// TIA Portal V20 export
DATA_BLOCK "HmiInterface"   // DB90
{ DB_Accessible_From_OPC_UA := 'FALSE' }
AUTHOR : ERsystem_FA2_DH. Kim
// stored: Access Published, DBAccessibleFromOPCUA false, DBAccessibleFromWebserver false, MemoryReserve 100, Namespace Unit1.Em4
   VAR
      em : "LAF_typeEmInterface";
      cm : Struct
         softCam : "Unit1.type_emRelations_em4_SoftCam";
         brakeTest : Struct
            anodeMainPnP1AxisZ : "LER_typeBrakeTestEmInterface";
            anodeMainPnP2AxisZ : "LER_typeBrakeTestEmInterface";
         END_STRUCT;
      END_STRUCT;
      mainPnP : Struct
         jobs { S7_SetPoint := 'True'} : "LAF_typeJobsInterface";
         sequence { S7_SetPoint := 'True'} : "LAF_typeSequenceInterface";
      END_STRUCT;
      alignTable : Struct
         jobs { S7_SetPoint := 'True'} : "LAF_typeJobsInterface";
         sequence { S7_SetPoint := 'True'} : "LAF_typeSequenceInterface";
      END_STRUCT;
      ngPnP : Struct
         jobs { S7_SetPoint := 'True'} : "LAF_typeJobsInterface";
         sequence { S7_SetPoint := 'True'} : "LAF_typeSequenceInterface";
      END_STRUCT;
      gaugeRnR : Struct
         jobs { S7_SetPoint := 'True'} : "LAF_typeJobsInterface";
         sequence { S7_SetPoint := 'True'} : "LAF_typeSequenceInterface";
      END_STRUCT;
      anodeNgCount : "LER_typeAlarmCounterInterface";
      cmPnp1stAnodeDetect { S7_SetPoint := 'True'} : "LBC_typeDigitalSignalInterface";
      cmPnp2ndAnodeDetect { S7_SetPoint := 'True'} : "LBC_typeDigitalSignalInterface";
      cmAnodeAlignTableElectrodeDetect { S7_SetPoint := 'True'} : "LBC_typeDigitalSignalInterface";
      cmAnodeNgPnpElectrodeDetect { S7_SetPoint := 'True'} : "LBC_typeDigitalSignalInterface";
      cmAnodeNgBoxFullSensorDetect { S7_SetPoint := 'True'} : "LBC_typeDigitalSignalInterface";
      cmAnodeNgBoxDetect { S7_SetPoint := 'True'} : "LBC_typeDigitalSignalInterface";
   END_VAR
   VAR RETAIN
      cmAnodeMainPnP1AxisX : "LBC_typeAxis64PosInterface";
      cmAnodeMainPnP2AxisX : "LBC_typeAxis64PosInterface";
      cmAnodeMainPnP1AxisY : "LBC_typeAxis64PosInterface";
      cmAnodeMainPnP1AxisZ : "LBC_typeAxis64PosInterface";
      cmAnodeMainPnP2AxisZ : "LBC_typeAxis64PosInterface";
      cmAnodeAlignTableAxisX : "LBC_typeAxis64PosInterface";
      cmAnodeAlignTableAxisY1 : "LBC_typeAxis64PosInterface";
      cmAnodeAlignTableAxisY2 : "LBC_typeAxis64PosInterface";
   END_VAR
   VAR
      cmAnodeMainPnP1RotaryCwCcw : "LBC_typeTwoWayActuatorInterface";
      cmAnodeMainPnP1SuctionPlateVacuum : "LBC_typeTwoWayActuatorInterface";
      cmAnodeMainPnP2SuctionPlateVacuum : "LBC_typeTwoWayActuatorInterface";
      cmAnodeAlignTableSuctionPlateVacuum : "LBC_typeTwoWayActuatorInterface";
      cmAnodeGlassCleaning : "LBC_typeTwoWayActuatorInterface";
      cmAnodeNgPnpUpDown : "LBC_typeTwoWayActuatorInterface";
      cmAnodeNgPnp1stFwdBwd : "LBC_typeTwoWayActuatorInterface";
      cmAnodeNgPnp2ndFwdBwd { S7_SetPoint := 'True'} : "LBC_typeTwoWayActuatorInterface";
      cmAnodeMaintenanceMovingFixFrontRearFwdBwd : "LBC_typeTwoWayActuatorInterface";
      cmAnodeNgBoxLiftUpDown { S7_SetPoint := 'True'} : "LBC_typeTwoWayActuatorInterface";
      cmAnodeNgBoxLockUpDown { S7_SetPoint := 'True'} : "LBC_typeTwoWayActuatorInterface";
      cmAnodeNgPnpVaccum : "LBC_typeTwoWayActuatorInterface";
      cmAnodeConveyorCoverFwdBwd { S7_SetPoint := 'True'} : "LBC_typeTwoWayActuatorInterface";
      cmAnodeConveyorPickUpBlower { S7_SetPoint := 'True'} : "LBC_typeTwoWayActuatorInterface";
      cmAlignVisionControllerInterface : "LER_typeVisionInterface";
      AlignVisionConversion : "LER_typeVisionAlignResultData";
      AlignMoveCalibration : "LER_typeAlignMoveCalibrationInterface";
      AlignThetaCalibration { S7_SetPoint := 'True'} : "LER_typeAlignThetaCalibrationInterface";
      AlignVisionHistory : "LER_typeVisionHistory";
      AlignSyncMove : "LER_typeAlignSyncMoveInterface";
      AlignCalibration : "LER_typeAlignCalibrationInterface";
   END_VAR
   VAR RETAIN
      GaugeRnR1Align : "LER_typeCount";
   END_VAR
   VAR
      GaugeRnR1Stack : "LER_typeCount";
      GaugeRnR3Align : "LER_typeCount";
      intCondition : Struct
         Axis_05 { S7_SetPoint := 'True'} : "LER.typeAxisIntlockAll";   // AnodeMainPnP1AxisX
         Axis_06 { S7_SetPoint := 'True'} : "LER.typeAxisIntlockAll";   // AnodeMainPnP2AxisX
         Axis_11 { S7_SetPoint := 'True'} : "LER.typeAxisIntlockAll";   // AnodeMainPnP1AxisY
         Axis_12 { S7_SetPoint := 'True'} : "LER.typeAxisIntlockAll";   // AnodeMainPnP1AxisZ
         Axis_14 { S7_SetPoint := 'True'} : "LER.typeAxisIntlockAll";   // AnodeMainPnP2AxisZ
         Axis_15 { S7_SetPoint := 'True'} : "LER.typeAxisIntlockAll";   // AnodeAlignTableAxisX
         Axis_16 { S7_SetPoint := 'True'} : "LER.typeAxisIntlockAll";   // AnodeAlignTableAxisY1
         Axis_17 { S7_SetPoint := 'True'} : "LER.typeAxisIntlockAll";   // AnodeAlignTableAxisY2
         Actuator_13 { S7_SetPoint := 'True'} : "LER.typeAxisActuatorCondition";   // AnodeNgBoxLiftUpDown
         Actuator_14 { S7_SetPoint := 'True'} : "LER.typeAxisActuatorCondition";   // SP
         Actuator_15 { S7_SetPoint := 'True'} : "LER.typeAxisActuatorCondition";   // AnodeNgBoxLockUpDown
         Actuator_16 { S7_SetPoint := 'True'} : "LER.typeAxisActuatorCondition";   // AnodeMaintenanceMovingFixFrontFwdBwd
         Actuator_17 { S7_SetPoint := 'True'} : "LER.typeAxisActuatorCondition";   // AnodeGlassCleaning
         Actuator_18 { S7_SetPoint := 'True'} : "LER.typeAxisActuatorCondition";   // AnodeNgPnp1stFwdBwd
         Actuator_19 { S7_SetPoint := 'True'} : "LER.typeAxisActuatorCondition";   // AnodeNgPnpUpDown
         Actuator_20 { S7_SetPoint := 'True'} : "LER.typeAxisActuatorCondition";   // SP
         Actuator_21 { S7_SetPoint := 'True'} : "LER.typeAxisActuatorCondition";   // AnodeMainPnP1RotaryCwCcw
         Actuator_22 { S7_SetPoint := 'True'} : "LER.typeAxisActuatorCondition";   // AnodeNgPnp2ndFwdBwd
      END_STRUCT;
   END_VAR
BEGIN
   em.interlinkMode.link := FALSE;
   em.interlinkMode.unlink := FALSE;
   em.interlinkMode.isLinked := TRUE;
   em.commands.enable := FALSE;
   em.commands.acknowledge := FALSE;
   em.commands.disableAlarms := FALSE;
   em.commands.activateSimulation := FALSE;
   em.commands.home := FALSE;
   em.commands.moveToInitialPosition := FALSE;
   em.commands.directModeControl := 16#0000_0001;
   em.commands.directStateControl := 16#0000_0004;
   em.status.enabled := TRUE;
   em.status.acknowledgeActive := FALSE;
   em.status.alarmsDisabled := FALSE;
   em.status.simulationActive := TRUE;
   em.status.safetyReleased := TRUE;
   em.status.initialized := FALSE;
   em.status.homed := FALSE;
   em.status.safeState := FALSE;
   em.status.stateComplete := FALSE;
   em.alarms.error := FALSE;
   em.alarms.warning := FALSE;
   em.alarms.info := FALSE;
   em.alarms.home := FALSE;
   cm.softCam.anodeMainPnP1AxisX.reelCutConveyerPos.inPos := TRUE;
   cm.softCam.anodeMainPnP1AxisX.reelCutConveyerPos.isBefore := FALSE;
   cm.softCam.anodeMainPnP1AxisX.reelCutConveyerPos.isAfter := FALSE;
   cm.softCam.anodeMainPnP1AxisX.alignTablePos.inPos := FALSE;
   cm.softCam.anodeMainPnP1AxisX.alignTablePos.isBefore := FALSE;
   cm.softCam.anodeMainPnP1AxisX.alignTablePos.isAfter := TRUE;
   cm.softCam.anodeMainPnP1AxisX.Pos2.inPos := FALSE;
   cm.softCam.anodeMainPnP1AxisX.Pos2.isBefore := FALSE;
   cm.softCam.anodeMainPnP1AxisX.Pos2.isAfter := TRUE;
   cm.softCam.anodeMainPnP1AxisX.Pos3.inPos := FALSE;
   cm.softCam.anodeMainPnP1AxisX.Pos3.isBefore := FALSE;
   cm.softCam.anodeMainPnP1AxisX.Pos3.isAfter := TRUE;
   cm.softCam.anodeMainPnP1AxisX.Pos4.inPos := FALSE;
   cm.softCam.anodeMainPnP1AxisX.Pos4.isBefore := FALSE;
   cm.softCam.anodeMainPnP1AxisX.Pos4.isAfter := TRUE;
   cm.softCam.anodeMainPnP1AxisX.Pos5.inPos := FALSE;
   cm.softCam.anodeMainPnP1AxisX.Pos5.isBefore := FALSE;
   cm.softCam.anodeMainPnP1AxisX.Pos5.isAfter := TRUE;
   cm.softCam.anodeMainPnP1AxisX.Pos6.inPos := FALSE;
   cm.softCam.anodeMainPnP1AxisX.Pos6.isBefore := FALSE;
   cm.softCam.anodeMainPnP1AxisX.Pos6.isAfter := TRUE;
   cm.softCam.anodeMainPnP1AxisX.Pos7.inPos := FALSE;
   cm.softCam.anodeMainPnP1AxisX.Pos7.isBefore := FALSE;
   cm.softCam.anodeMainPnP1AxisX.Pos7.isAfter := TRUE;
   cm.softCam.anodeMainPnP1AxisX.Pos8.inPos := FALSE;
   cm.softCam.anodeMainPnP1AxisX.Pos8.isBefore := FALSE;
   cm.softCam.anodeMainPnP1AxisX.Pos8.isAfter := TRUE;
   cm.softCam.anodeMainPnP1AxisX.Pos9.inPos := FALSE;
   cm.softCam.anodeMainPnP1AxisX.Pos9.isBefore := FALSE;
   cm.softCam.anodeMainPnP1AxisX.Pos9.isAfter := TRUE;
   cm.softCam.anodeMainPnP1AxisX.Pos10.inPos := FALSE;
   cm.softCam.anodeMainPnP1AxisX.Pos10.isBefore := FALSE;
   cm.softCam.anodeMainPnP1AxisX.Pos10.isAfter := TRUE;
   cm.softCam.anodeMainPnP1AxisX.Pos11.inPos := FALSE;
   cm.softCam.anodeMainPnP1AxisX.Pos11.isBefore := FALSE;
   cm.softCam.anodeMainPnP1AxisX.Pos11.isAfter := TRUE;
   cm.softCam.anodeMainPnP1AxisX.Pos12.inPos := FALSE;
   cm.softCam.anodeMainPnP1AxisX.Pos12.isBefore := FALSE;
   cm.softCam.anodeMainPnP1AxisX.Pos12.isAfter := TRUE;
   cm.softCam.anodeMainPnP1AxisX.Pos13.inPos := FALSE;
   cm.softCam.anodeMainPnP1AxisX.Pos13.isBefore := FALSE;
   cm.softCam.anodeMainPnP1AxisX.Pos13.isAfter := TRUE;
   cm.softCam.anodeMainPnP1AxisX.Pos14.inPos := FALSE;
   cm.softCam.anodeMainPnP1AxisX.Pos14.isBefore := FALSE;
   cm.softCam.anodeMainPnP1AxisX.Pos14.isAfter := TRUE;
   cm.softCam.anodeMainPnP1AxisX.Pos15.inPos := FALSE;
   cm.softCam.anodeMainPnP1AxisX.Pos15.isBefore := FALSE;
   cm.softCam.anodeMainPnP1AxisX.Pos15.isAfter := TRUE;
   cm.softCam.anodeMainPnP2AxisX.alignTablePos.inPos := TRUE;
   cm.softCam.anodeMainPnP2AxisX.alignTablePos.isBefore := FALSE;
   cm.softCam.anodeMainPnP2AxisX.alignTablePos.isAfter := FALSE;
   cm.softCam.anodeMainPnP2AxisX.stackTablePos.inPos := FALSE;
   cm.softCam.anodeMainPnP2AxisX.stackTablePos.isBefore := FALSE;
   cm.softCam.anodeMainPnP2AxisX.stackTablePos.isAfter := TRUE;
   cm.softCam.anodeMainPnP2AxisX.Pos2.inPos := FALSE;
   cm.softCam.anodeMainPnP2AxisX.Pos2.isBefore := FALSE;
   cm.softCam.anodeMainPnP2AxisX.Pos2.isAfter := TRUE;
   cm.softCam.anodeMainPnP2AxisX.Pos3.inPos := FALSE;
   cm.softCam.anodeMainPnP2AxisX.Pos3.isBefore := FALSE;
   cm.softCam.anodeMainPnP2AxisX.Pos3.isAfter := TRUE;
   cm.softCam.anodeMainPnP2AxisX.Pos4.inPos := FALSE;
   cm.softCam.anodeMainPnP2AxisX.Pos4.isBefore := FALSE;
   cm.softCam.anodeMainPnP2AxisX.Pos4.isAfter := TRUE;
   cm.softCam.anodeMainPnP2AxisX.Pos5.inPos := FALSE;
   cm.softCam.anodeMainPnP2AxisX.Pos5.isBefore := FALSE;
   cm.softCam.anodeMainPnP2AxisX.Pos5.isAfter := TRUE;
   cm.softCam.anodeMainPnP2AxisX.Pos6.inPos := FALSE;
   cm.softCam.anodeMainPnP2AxisX.Pos6.isBefore := FALSE;
   cm.softCam.anodeMainPnP2AxisX.Pos6.isAfter := TRUE;
   cm.softCam.anodeMainPnP2AxisX.Pos7.inPos := FALSE;
   cm.softCam.anodeMainPnP2AxisX.Pos7.isBefore := FALSE;
   cm.softCam.anodeMainPnP2AxisX.Pos7.isAfter := TRUE;
   cm.softCam.anodeMainPnP2AxisX.Pos8.inPos := FALSE;
   cm.softCam.anodeMainPnP2AxisX.Pos8.isBefore := FALSE;
   cm.softCam.anodeMainPnP2AxisX.Pos8.isAfter := TRUE;
   cm.softCam.anodeMainPnP2AxisX.Pos9.inPos := FALSE;
   cm.softCam.anodeMainPnP2AxisX.Pos9.isBefore := FALSE;
   cm.softCam.anodeMainPnP2AxisX.Pos9.isAfter := TRUE;
   cm.softCam.anodeMainPnP2AxisX.Pos10.inPos := FALSE;
   cm.softCam.anodeMainPnP2AxisX.Pos10.isBefore := FALSE;
   cm.softCam.anodeMainPnP2AxisX.Pos10.isAfter := TRUE;
   cm.softCam.anodeMainPnP2AxisX.Pos11.inPos := FALSE;
   cm.softCam.anodeMainPnP2AxisX.Pos11.isBefore := FALSE;
   cm.softCam.anodeMainPnP2AxisX.Pos11.isAfter := TRUE;
   cm.softCam.anodeMainPnP2AxisX.Pos12.inPos := FALSE;
   cm.softCam.anodeMainPnP2AxisX.Pos12.isBefore := FALSE;
   cm.softCam.anodeMainPnP2AxisX.Pos12.isAfter := TRUE;
   cm.softCam.anodeMainPnP2AxisX.Pos13.inPos := FALSE;
   cm.softCam.anodeMainPnP2AxisX.Pos13.isBefore := FALSE;
   cm.softCam.anodeMainPnP2AxisX.Pos13.isAfter := TRUE;
   cm.softCam.anodeMainPnP2AxisX.Pos14.inPos := FALSE;
   cm.softCam.anodeMainPnP2AxisX.Pos14.isBefore := FALSE;
   cm.softCam.anodeMainPnP2AxisX.Pos14.isAfter := TRUE;
   cm.softCam.anodeMainPnP2AxisX.Pos15.inPos := FALSE;
   cm.softCam.anodeMainPnP2AxisX.Pos15.isBefore := FALSE;
   cm.softCam.anodeMainPnP2AxisX.Pos15.isAfter := TRUE;
   cm.softCam.anodeMainPnP1AxisY.waitPos.inPos := TRUE;
   cm.softCam.anodeMainPnP1AxisY.waitPos.isBefore := FALSE;
   cm.softCam.anodeMainPnP1AxisY.waitPos.isAfter := FALSE;
   cm.softCam.anodeMainPnP1AxisY.Pos1.inPos := TRUE;
   cm.softCam.anodeMainPnP1AxisY.Pos1.isBefore := FALSE;
   cm.softCam.anodeMainPnP1AxisY.Pos1.isAfter := FALSE;
   cm.softCam.anodeMainPnP1AxisY.Pos2.inPos := TRUE;
   cm.softCam.anodeMainPnP1AxisY.Pos2.isBefore := FALSE;
   cm.softCam.anodeMainPnP1AxisY.Pos2.isAfter := FALSE;
   cm.softCam.anodeMainPnP1AxisY.Pos3.inPos := TRUE;
   cm.softCam.anodeMainPnP1AxisY.Pos3.isBefore := FALSE;
   cm.softCam.anodeMainPnP1AxisY.Pos3.isAfter := FALSE;
   cm.softCam.anodeMainPnP1AxisY.Pos4.inPos := TRUE;
   cm.softCam.anodeMainPnP1AxisY.Pos4.isBefore := FALSE;
   cm.softCam.anodeMainPnP1AxisY.Pos4.isAfter := FALSE;
   cm.softCam.anodeMainPnP1AxisY.Pos5.inPos := TRUE;
   cm.softCam.anodeMainPnP1AxisY.Pos5.isBefore := FALSE;
   cm.softCam.anodeMainPnP1AxisY.Pos5.isAfter := FALSE;
   cm.softCam.anodeMainPnP1AxisY.Pos6.inPos := TRUE;
   cm.softCam.anodeMainPnP1AxisY.Pos6.isBefore := FALSE;
   cm.softCam.anodeMainPnP1AxisY.Pos6.isAfter := FALSE;
   cm.softCam.anodeMainPnP1AxisY.Pos7.inPos := TRUE;
   cm.softCam.anodeMainPnP1AxisY.Pos7.isBefore := FALSE;
   cm.softCam.anodeMainPnP1AxisY.Pos7.isAfter := FALSE;
   cm.softCam.anodeMainPnP1AxisY.Pos8.inPos := TRUE;
   cm.softCam.anodeMainPnP1AxisY.Pos8.isBefore := FALSE;
   cm.softCam.anodeMainPnP1AxisY.Pos8.isAfter := FALSE;
   cm.softCam.anodeMainPnP1AxisY.Pos9.inPos := TRUE;
   cm.softCam.anodeMainPnP1AxisY.Pos9.isBefore := FALSE;
   cm.softCam.anodeMainPnP1AxisY.Pos9.isAfter := FALSE;
   cm.softCam.anodeMainPnP1AxisY.Pos10.inPos := TRUE;
   cm.softCam.anodeMainPnP1AxisY.Pos10.isBefore := FALSE;
   cm.softCam.anodeMainPnP1AxisY.Pos10.isAfter := FALSE;
   cm.softCam.anodeMainPnP1AxisY.Pos11.inPos := TRUE;
   cm.softCam.anodeMainPnP1AxisY.Pos11.isBefore := FALSE;
   cm.softCam.anodeMainPnP1AxisY.Pos11.isAfter := FALSE;
   cm.softCam.anodeMainPnP1AxisY.Pos12.inPos := TRUE;
   cm.softCam.anodeMainPnP1AxisY.Pos12.isBefore := FALSE;
   cm.softCam.anodeMainPnP1AxisY.Pos12.isAfter := FALSE;
   cm.softCam.anodeMainPnP1AxisY.Pos13.inPos := TRUE;
   cm.softCam.anodeMainPnP1AxisY.Pos13.isBefore := FALSE;
   cm.softCam.anodeMainPnP1AxisY.Pos13.isAfter := FALSE;
   cm.softCam.anodeMainPnP1AxisY.Pos14.inPos := TRUE;
   cm.softCam.anodeMainPnP1AxisY.Pos14.isBefore := FALSE;
   cm.softCam.anodeMainPnP1AxisY.Pos14.isAfter := FALSE;
   cm.softCam.anodeMainPnP1AxisY.Pos15.inPos := TRUE;
   cm.softCam.anodeMainPnP1AxisY.Pos15.isBefore := FALSE;
   cm.softCam.anodeMainPnP1AxisY.Pos15.isAfter := FALSE;
   cm.softCam.anodeMainPnP1AxisZ.upPos.inPos := FALSE;
   cm.softCam.anodeMainPnP1AxisZ.upPos.isBefore := FALSE;
   cm.softCam.anodeMainPnP1AxisZ.upPos.isAfter := TRUE;
   cm.softCam.anodeMainPnP1AxisZ.reelCutConveyerDownPos.inPos := TRUE;
   cm.softCam.anodeMainPnP1AxisZ.reelCutConveyerDownPos.isBefore := FALSE;
   cm.softCam.anodeMainPnP1AxisZ.reelCutConveyerDownPos.isAfter := FALSE;
   cm.softCam.anodeMainPnP1AxisZ.ailgnTableDownPos.inPos := TRUE;
   cm.softCam.anodeMainPnP1AxisZ.ailgnTableDownPos.isBefore := FALSE;
   cm.softCam.anodeMainPnP1AxisZ.ailgnTableDownPos.isAfter := FALSE;
   cm.softCam.anodeMainPnP1AxisZ.avoidPos.inPos := FALSE;
   cm.softCam.anodeMainPnP1AxisZ.avoidPos.isBefore := FALSE;
   cm.softCam.anodeMainPnP1AxisZ.avoidPos.isAfter := TRUE;
   cm.softCam.anodeMainPnP1AxisZ.Pos4.inPos := FALSE;
   cm.softCam.anodeMainPnP1AxisZ.Pos4.isBefore := FALSE;
   cm.softCam.anodeMainPnP1AxisZ.Pos4.isAfter := TRUE;
   cm.softCam.anodeMainPnP1AxisZ.Pos5.inPos := FALSE;
   cm.softCam.anodeMainPnP1AxisZ.Pos5.isBefore := FALSE;
   cm.softCam.anodeMainPnP1AxisZ.Pos5.isAfter := TRUE;
   cm.softCam.anodeMainPnP1AxisZ.Pos6.inPos := FALSE;
   cm.softCam.anodeMainPnP1AxisZ.Pos6.isBefore := FALSE;
   cm.softCam.anodeMainPnP1AxisZ.Pos6.isAfter := TRUE;
   cm.softCam.anodeMainPnP1AxisZ.Pos7.inPos := FALSE;
   cm.softCam.anodeMainPnP1AxisZ.Pos7.isBefore := FALSE;
   cm.softCam.anodeMainPnP1AxisZ.Pos7.isAfter := TRUE;
   cm.softCam.anodeMainPnP1AxisZ.Pos8.inPos := FALSE;
   cm.softCam.anodeMainPnP1AxisZ.Pos8.isBefore := FALSE;
   cm.softCam.anodeMainPnP1AxisZ.Pos8.isAfter := TRUE;
   cm.softCam.anodeMainPnP1AxisZ.Pos9.inPos := FALSE;
   cm.softCam.anodeMainPnP1AxisZ.Pos9.isBefore := FALSE;
   cm.softCam.anodeMainPnP1AxisZ.Pos9.isAfter := TRUE;
   cm.softCam.anodeMainPnP1AxisZ.Pos10.inPos := FALSE;
   cm.softCam.anodeMainPnP1AxisZ.Pos10.isBefore := FALSE;
   cm.softCam.anodeMainPnP1AxisZ.Pos10.isAfter := TRUE;
   cm.softCam.anodeMainPnP1AxisZ.Pos11.inPos := FALSE;
   cm.softCam.anodeMainPnP1AxisZ.Pos11.isBefore := FALSE;
   cm.softCam.anodeMainPnP1AxisZ.Pos11.isAfter := TRUE;
   cm.softCam.anodeMainPnP1AxisZ.Pos12.inPos := FALSE;
   cm.softCam.anodeMainPnP1AxisZ.Pos12.isBefore := FALSE;
   cm.softCam.anodeMainPnP1AxisZ.Pos12.isAfter := TRUE;
   cm.softCam.anodeMainPnP1AxisZ.Pos13.inPos := FALSE;
   cm.softCam.anodeMainPnP1AxisZ.Pos13.isBefore := FALSE;
   cm.softCam.anodeMainPnP1AxisZ.Pos13.isAfter := TRUE;
   cm.softCam.anodeMainPnP1AxisZ.Pos14.inPos := FALSE;
   cm.softCam.anodeMainPnP1AxisZ.Pos14.isBefore := FALSE;
   cm.softCam.anodeMainPnP1AxisZ.Pos14.isAfter := TRUE;
   cm.softCam.anodeMainPnP1AxisZ.Pos15.inPos := FALSE;
   cm.softCam.anodeMainPnP1AxisZ.Pos15.isBefore := FALSE;
   cm.softCam.anodeMainPnP1AxisZ.Pos15.isAfter := TRUE;
   cm.softCam.anodeMainPnP2AxisZ.upPos.inPos := FALSE;
   cm.softCam.anodeMainPnP2AxisZ.upPos.isBefore := FALSE;
   cm.softCam.anodeMainPnP2AxisZ.upPos.isAfter := TRUE;
   cm.softCam.anodeMainPnP2AxisZ.ailgnTableDownPos.inPos := TRUE;
   cm.softCam.anodeMainPnP2AxisZ.ailgnTableDownPos.isBefore := FALSE;
   cm.softCam.anodeMainPnP2AxisZ.ailgnTableDownPos.isAfter := FALSE;
   cm.softCam.anodeMainPnP2AxisZ.stackTableDownPos.inPos := TRUE;
   cm.softCam.anodeMainPnP2AxisZ.stackTableDownPos.isBefore := FALSE;
   cm.softCam.anodeMainPnP2AxisZ.stackTableDownPos.isAfter := FALSE;
   cm.softCam.anodeMainPnP2AxisZ.avoidPos.inPos := FALSE;
   cm.softCam.anodeMainPnP2AxisZ.avoidPos.isBefore := FALSE;
   cm.softCam.anodeMainPnP2AxisZ.avoidPos.isAfter := TRUE;
   cm.softCam.anodeMainPnP2AxisZ.Pos4.inPos := FALSE;
   cm.softCam.anodeMainPnP2AxisZ.Pos4.isBefore := FALSE;
   cm.softCam.anodeMainPnP2AxisZ.Pos4.isAfter := TRUE;
   cm.softCam.anodeMainPnP2AxisZ.Pos5.inPos := FALSE;
   cm.softCam.anodeMainPnP2AxisZ.Pos5.isBefore := FALSE;
   cm.softCam.anodeMainPnP2AxisZ.Pos5.isAfter := TRUE;
   cm.softCam.anodeMainPnP2AxisZ.Pos6.inPos := FALSE;
   cm.softCam.anodeMainPnP2AxisZ.Pos6.isBefore := FALSE;
   cm.softCam.anodeMainPnP2AxisZ.Pos6.isAfter := TRUE;
   cm.softCam.anodeMainPnP2AxisZ.Pos7.inPos := FALSE;
   cm.softCam.anodeMainPnP2AxisZ.Pos7.isBefore := FALSE;
   cm.softCam.anodeMainPnP2AxisZ.Pos7.isAfter := TRUE;
   cm.softCam.anodeMainPnP2AxisZ.Pos8.inPos := FALSE;
   cm.softCam.anodeMainPnP2AxisZ.Pos8.isBefore := FALSE;
   cm.softCam.anodeMainPnP2AxisZ.Pos8.isAfter := TRUE;
   cm.softCam.anodeMainPnP2AxisZ.Pos9.inPos := FALSE;
   cm.softCam.anodeMainPnP2AxisZ.Pos9.isBefore := FALSE;
   cm.softCam.anodeMainPnP2AxisZ.Pos9.isAfter := TRUE;
   cm.softCam.anodeMainPnP2AxisZ.Pos10.inPos := FALSE;
   cm.softCam.anodeMainPnP2AxisZ.Pos10.isBefore := FALSE;
   cm.softCam.anodeMainPnP2AxisZ.Pos10.isAfter := TRUE;
   cm.softCam.anodeMainPnP2AxisZ.Pos11.inPos := FALSE;
   cm.softCam.anodeMainPnP2AxisZ.Pos11.isBefore := FALSE;
   cm.softCam.anodeMainPnP2AxisZ.Pos11.isAfter := TRUE;
   cm.softCam.anodeMainPnP2AxisZ.Pos12.inPos := FALSE;
   cm.softCam.anodeMainPnP2AxisZ.Pos12.isBefore := FALSE;
   cm.softCam.anodeMainPnP2AxisZ.Pos12.isAfter := TRUE;
   cm.softCam.anodeMainPnP2AxisZ.Pos13.inPos := FALSE;
   cm.softCam.anodeMainPnP2AxisZ.Pos13.isBefore := FALSE;
   cm.softCam.anodeMainPnP2AxisZ.Pos13.isAfter := TRUE;
   cm.softCam.anodeMainPnP2AxisZ.Pos14.inPos := FALSE;
   cm.softCam.anodeMainPnP2AxisZ.Pos14.isBefore := FALSE;
   cm.softCam.anodeMainPnP2AxisZ.Pos14.isAfter := TRUE;
   cm.softCam.anodeMainPnP2AxisZ.Pos15.inPos := FALSE;
   cm.softCam.anodeMainPnP2AxisZ.Pos15.isBefore := FALSE;
   cm.softCam.anodeMainPnP2AxisZ.Pos15.isAfter := TRUE;
   cm.softCam.anodeAlignTableAxisX.waitPos.inPos := TRUE;
   cm.softCam.anodeAlignTableAxisX.waitPos.isBefore := FALSE;
   cm.softCam.anodeAlignTableAxisX.waitPos.isAfter := FALSE;
   cm.softCam.anodeAlignTableAxisX.adjustPos.inPos := FALSE;
   cm.softCam.anodeAlignTableAxisX.adjustPos.isBefore := TRUE;
   cm.softCam.anodeAlignTableAxisX.adjustPos.isAfter := FALSE;
   cm.softCam.anodeAlignTableAxisX.Pos2.inPos := FALSE;
   cm.softCam.anodeAlignTableAxisX.Pos2.isBefore := FALSE;
   cm.softCam.anodeAlignTableAxisX.Pos2.isAfter := TRUE;
   cm.softCam.anodeAlignTableAxisX.Pos3.inPos := FALSE;
   cm.softCam.anodeAlignTableAxisX.Pos3.isBefore := FALSE;
   cm.softCam.anodeAlignTableAxisX.Pos3.isAfter := TRUE;
   cm.softCam.anodeAlignTableAxisX.Pos4.inPos := FALSE;
   cm.softCam.anodeAlignTableAxisX.Pos4.isBefore := FALSE;
   cm.softCam.anodeAlignTableAxisX.Pos4.isAfter := TRUE;
   cm.softCam.anodeAlignTableAxisX.Pos5.inPos := FALSE;
   cm.softCam.anodeAlignTableAxisX.Pos5.isBefore := FALSE;
   cm.softCam.anodeAlignTableAxisX.Pos5.isAfter := TRUE;
   cm.softCam.anodeAlignTableAxisX.Pos6.inPos := FALSE;
   cm.softCam.anodeAlignTableAxisX.Pos6.isBefore := FALSE;
   cm.softCam.anodeAlignTableAxisX.Pos6.isAfter := TRUE;
   cm.softCam.anodeAlignTableAxisX.Pos7.inPos := FALSE;
   cm.softCam.anodeAlignTableAxisX.Pos7.isBefore := FALSE;
   cm.softCam.anodeAlignTableAxisX.Pos7.isAfter := TRUE;
   cm.softCam.anodeAlignTableAxisX.Pos8.inPos := FALSE;
   cm.softCam.anodeAlignTableAxisX.Pos8.isBefore := FALSE;
   cm.softCam.anodeAlignTableAxisX.Pos8.isAfter := TRUE;
   cm.softCam.anodeAlignTableAxisX.Pos9.inPos := FALSE;
   cm.softCam.anodeAlignTableAxisX.Pos9.isBefore := FALSE;
   cm.softCam.anodeAlignTableAxisX.Pos9.isAfter := TRUE;
   cm.softCam.anodeAlignTableAxisX.Pos10.inPos := FALSE;
   cm.softCam.anodeAlignTableAxisX.Pos10.isBefore := TRUE;
   cm.softCam.anodeAlignTableAxisX.Pos10.isAfter := FALSE;
   cm.softCam.anodeAlignTableAxisX.Pos11.inPos := TRUE;
   cm.softCam.anodeAlignTableAxisX.Pos11.isBefore := FALSE;
   cm.softCam.anodeAlignTableAxisX.Pos11.isAfter := FALSE;
   cm.softCam.anodeAlignTableAxisX.Pos12.inPos := TRUE;
   cm.softCam.anodeAlignTableAxisX.Pos12.isBefore := FALSE;
   cm.softCam.anodeAlignTableAxisX.Pos12.isAfter := FALSE;
   cm.softCam.anodeAlignTableAxisX.Pos13.inPos := TRUE;
   cm.softCam.anodeAlignTableAxisX.Pos13.isBefore := FALSE;
   cm.softCam.anodeAlignTableAxisX.Pos13.isAfter := FALSE;
   cm.softCam.anodeAlignTableAxisX.Pos14.inPos := TRUE;
   cm.softCam.anodeAlignTableAxisX.Pos14.isBefore := FALSE;
   cm.softCam.anodeAlignTableAxisX.Pos14.isAfter := FALSE;
   cm.softCam.anodeAlignTableAxisX.Pos15.inPos := TRUE;
   cm.softCam.anodeAlignTableAxisX.Pos15.isBefore := FALSE;
   cm.softCam.anodeAlignTableAxisX.Pos15.isAfter := FALSE;
   cm.softCam.anodeAlignTableAxisY1.waitPos.inPos := TRUE;
   cm.softCam.anodeAlignTableAxisY1.waitPos.isBefore := FALSE;
   cm.softCam.anodeAlignTableAxisY1.waitPos.isAfter := FALSE;
   cm.softCam.anodeAlignTableAxisY1.adjustPos.inPos := FALSE;
   cm.softCam.anodeAlignTableAxisY1.adjustPos.isBefore := TRUE;
   cm.softCam.anodeAlignTableAxisY1.adjustPos.isAfter := FALSE;
   cm.softCam.anodeAlignTableAxisY1.Pos2.inPos := FALSE;
   cm.softCam.anodeAlignTableAxisY1.Pos2.isBefore := TRUE;
   cm.softCam.anodeAlignTableAxisY1.Pos2.isAfter := FALSE;
   cm.softCam.anodeAlignTableAxisY1.Pos3.inPos := FALSE;
   cm.softCam.anodeAlignTableAxisY1.Pos3.isBefore := TRUE;
   cm.softCam.anodeAlignTableAxisY1.Pos3.isAfter := FALSE;
   cm.softCam.anodeAlignTableAxisY1.Pos4.inPos := FALSE;
   cm.softCam.anodeAlignTableAxisY1.Pos4.isBefore := TRUE;
   cm.softCam.anodeAlignTableAxisY1.Pos4.isAfter := FALSE;
   cm.softCam.anodeAlignTableAxisY1.Pos5.inPos := FALSE;
   cm.softCam.anodeAlignTableAxisY1.Pos5.isBefore := TRUE;
   cm.softCam.anodeAlignTableAxisY1.Pos5.isAfter := FALSE;
   cm.softCam.anodeAlignTableAxisY1.Pos6.inPos := FALSE;
   cm.softCam.anodeAlignTableAxisY1.Pos6.isBefore := TRUE;
   cm.softCam.anodeAlignTableAxisY1.Pos6.isAfter := FALSE;
   cm.softCam.anodeAlignTableAxisY1.Pos7.inPos := FALSE;
   cm.softCam.anodeAlignTableAxisY1.Pos7.isBefore := FALSE;
   cm.softCam.anodeAlignTableAxisY1.Pos7.isAfter := TRUE;
   cm.softCam.anodeAlignTableAxisY1.Pos8.inPos := FALSE;
   cm.softCam.anodeAlignTableAxisY1.Pos8.isBefore := TRUE;
   cm.softCam.anodeAlignTableAxisY1.Pos8.isAfter := FALSE;
   cm.softCam.anodeAlignTableAxisY1.Pos9.inPos := FALSE;
   cm.softCam.anodeAlignTableAxisY1.Pos9.isBefore := FALSE;
   cm.softCam.anodeAlignTableAxisY1.Pos9.isAfter := TRUE;
   cm.softCam.anodeAlignTableAxisY1.Pos10.inPos := FALSE;
   cm.softCam.anodeAlignTableAxisY1.Pos10.isBefore := TRUE;
   cm.softCam.anodeAlignTableAxisY1.Pos10.isAfter := FALSE;
   cm.softCam.anodeAlignTableAxisY1.Pos11.inPos := TRUE;
   cm.softCam.anodeAlignTableAxisY1.Pos11.isBefore := FALSE;
   cm.softCam.anodeAlignTableAxisY1.Pos11.isAfter := FALSE;
   cm.softCam.anodeAlignTableAxisY1.Pos12.inPos := TRUE;
   cm.softCam.anodeAlignTableAxisY1.Pos12.isBefore := FALSE;
   cm.softCam.anodeAlignTableAxisY1.Pos12.isAfter := FALSE;
   cm.softCam.anodeAlignTableAxisY1.Pos13.inPos := TRUE;
   cm.softCam.anodeAlignTableAxisY1.Pos13.isBefore := FALSE;
   cm.softCam.anodeAlignTableAxisY1.Pos13.isAfter := FALSE;
   cm.softCam.anodeAlignTableAxisY1.Pos14.inPos := TRUE;
   cm.softCam.anodeAlignTableAxisY1.Pos14.isBefore := FALSE;
   cm.softCam.anodeAlignTableAxisY1.Pos14.isAfter := FALSE;
   cm.softCam.anodeAlignTableAxisY1.Pos15.inPos := TRUE;
   cm.softCam.anodeAlignTableAxisY1.Pos15.isBefore := FALSE;
   cm.softCam.anodeAlignTableAxisY1.Pos15.isAfter := FALSE;
   cm.softCam.anodeAlignTableAxisY2.waitPos.inPos := TRUE;
   cm.softCam.anodeAlignTableAxisY2.waitPos.isBefore := FALSE;
   cm.softCam.anodeAlignTableAxisY2.waitPos.isAfter := FALSE;
   cm.softCam.anodeAlignTableAxisY2.adjustPos.inPos := FALSE;
   cm.softCam.anodeAlignTableAxisY2.adjustPos.isBefore := TRUE;
   cm.softCam.anodeAlignTableAxisY2.adjustPos.isAfter := FALSE;
   cm.softCam.anodeAlignTableAxisY2.Pos2.inPos := TRUE;
   cm.softCam.anodeAlignTableAxisY2.Pos2.isBefore := FALSE;
   cm.softCam.anodeAlignTableAxisY2.Pos2.isAfter := FALSE;
   cm.softCam.anodeAlignTableAxisY2.Pos3.inPos := TRUE;
   cm.softCam.anodeAlignTableAxisY2.Pos3.isBefore := FALSE;
   cm.softCam.anodeAlignTableAxisY2.Pos3.isAfter := FALSE;
   cm.softCam.anodeAlignTableAxisY2.Pos4.inPos := TRUE;
   cm.softCam.anodeAlignTableAxisY2.Pos4.isBefore := FALSE;
   cm.softCam.anodeAlignTableAxisY2.Pos4.isAfter := FALSE;
   cm.softCam.anodeAlignTableAxisY2.Pos5.inPos := TRUE;
   cm.softCam.anodeAlignTableAxisY2.Pos5.isBefore := FALSE;
   cm.softCam.anodeAlignTableAxisY2.Pos5.isAfter := FALSE;
   cm.softCam.anodeAlignTableAxisY2.Pos6.inPos := TRUE;
   cm.softCam.anodeAlignTableAxisY2.Pos6.isBefore := FALSE;
   cm.softCam.anodeAlignTableAxisY2.Pos6.isAfter := FALSE;
   cm.softCam.anodeAlignTableAxisY2.Pos7.inPos := TRUE;
   cm.softCam.anodeAlignTableAxisY2.Pos7.isBefore := FALSE;
   cm.softCam.anodeAlignTableAxisY2.Pos7.isAfter := FALSE;
   cm.softCam.anodeAlignTableAxisY2.Pos8.inPos := TRUE;
   cm.softCam.anodeAlignTableAxisY2.Pos8.isBefore := FALSE;
   cm.softCam.anodeAlignTableAxisY2.Pos8.isAfter := FALSE;
   cm.softCam.anodeAlignTableAxisY2.Pos9.inPos := TRUE;
   cm.softCam.anodeAlignTableAxisY2.Pos9.isBefore := FALSE;
   cm.softCam.anodeAlignTableAxisY2.Pos9.isAfter := FALSE;
   cm.softCam.anodeAlignTableAxisY2.Pos10.inPos := FALSE;
   cm.softCam.anodeAlignTableAxisY2.Pos10.isBefore := TRUE;
   cm.softCam.anodeAlignTableAxisY2.Pos10.isAfter := FALSE;
   cm.softCam.anodeAlignTableAxisY2.Pos11.inPos := TRUE;
   cm.softCam.anodeAlignTableAxisY2.Pos11.isBefore := FALSE;
   cm.softCam.anodeAlignTableAxisY2.Pos11.isAfter := FALSE;
   cm.softCam.anodeAlignTableAxisY2.Pos12.inPos := TRUE;
   cm.softCam.anodeAlignTableAxisY2.Pos12.isBefore := FALSE;
   cm.softCam.anodeAlignTableAxisY2.Pos12.isAfter := FALSE;
   cm.softCam.anodeAlignTableAxisY2.Pos13.inPos := TRUE;
   cm.softCam.anodeAlignTableAxisY2.Pos13.isBefore := FALSE;
   cm.softCam.anodeAlignTableAxisY2.Pos13.isAfter := FALSE;
   cm.softCam.anodeAlignTableAxisY2.Pos14.inPos := TRUE;
   cm.softCam.anodeAlignTableAxisY2.Pos14.isBefore := FALSE;
   cm.softCam.anodeAlignTableAxisY2.Pos14.isAfter := FALSE;
   cm.softCam.anodeAlignTableAxisY2.Pos15.inPos := TRUE;
   cm.softCam.anodeAlignTableAxisY2.Pos15.isBefore := FALSE;
   cm.softCam.anodeAlignTableAxisY2.Pos15.isAfter := FALSE;
   cm.brakeTest.anodeMainPnP1AxisZ.commands.start := FALSE;
   cm.brakeTest.anodeMainPnP1AxisZ.commands.stop := FALSE;
   cm.brakeTest.anodeMainPnP1AxisZ.monitoring.error := FALSE;
   cm.brakeTest.anodeMainPnP1AxisZ.monitoring.ready := FALSE;
   cm.brakeTest.anodeMainPnP1AxisZ.monitoring.busy := FALSE;
   cm.brakeTest.anodeMainPnP1AxisZ.monitoring.complete := FALSE;
   cm.brakeTest.anodeMainPnP1AxisZ.monitoring.brakeSelected := FALSE;
   cm.brakeTest.anodeMainPnP1AxisZ.monitoring.brakeActive := FALSE;
   cm.brakeTest.anodeMainPnP1AxisZ.monitoring.brakeResult := FALSE;
   cm.brakeTest.anodeMainPnP1AxisZ.monitoring.brakeCompleted := FALSE;
   cm.brakeTest.anodeMainPnP1AxisZ.monitoring."step" := 0;
   cm.brakeTest.anodeMainPnP2AxisZ.commands.start := FALSE;
   cm.brakeTest.anodeMainPnP2AxisZ.commands.stop := FALSE;
   cm.brakeTest.anodeMainPnP2AxisZ.monitoring.error := FALSE;
   cm.brakeTest.anodeMainPnP2AxisZ.monitoring.ready := FALSE;
   cm.brakeTest.anodeMainPnP2AxisZ.monitoring.busy := FALSE;
   cm.brakeTest.anodeMainPnP2AxisZ.monitoring.complete := FALSE;
   cm.brakeTest.anodeMainPnP2AxisZ.monitoring.brakeSelected := FALSE;
   cm.brakeTest.anodeMainPnP2AxisZ.monitoring.brakeActive := FALSE;
   cm.brakeTest.anodeMainPnP2AxisZ.monitoring.brakeResult := FALSE;
   cm.brakeTest.anodeMainPnP2AxisZ.monitoring.brakeCompleted := FALSE;
   cm.brakeTest.anodeMainPnP2AxisZ.monitoring."step" := 0;
   mainPnP.jobs.commands.setJobNumber := 0;
   mainPnP.jobs.commands.reset := FALSE;
   mainPnP.jobs.status.activeJobNumber := 0;
   mainPnP.jobs.status.previousCycleJobNumber := 0;
   mainPnP.jobs.status.manualControlEnabled := FALSE;
   mainPnP.jobs.status.memoryJobTime := 16#0000_4EB7_0DCE_2E62;
   mainPnP.sequence.commands.setAutomaticMode := FALSE;
   mainPnP.sequence.commands.setSingleStepMode := FALSE;
   mainPnP.sequence.commands.off := FALSE;
   mainPnP.sequence.commands.initialize := FALSE;
   mainPnP.sequence.commands.start := FALSE;
   mainPnP.sequence.commands.immediateStop := FALSE;
   mainPnP.sequence.commands.hold := FALSE;
   mainPnP.sequence.commands.nextStep := FALSE;
   mainPnP.sequence.commands.interlockStepChange := FALSE;
   mainPnP.sequence.monitoring.automaticMode := TRUE;
   mainPnP.sequence.monitoring.singleStepMode := FALSE;
   mainPnP.sequence.monitoring.currentStep := 1;
   mainPnP.sequence.monitoring.nextStep := 1;
   mainPnP.sequence.monitoring.previousStep := 190;
   mainPnP.sequence.monitoring.currentStepSTRING := 'N/A';
   mainPnP.sequence.monitoring.nextStepSTRING := 'N/A';
   mainPnP.sequence.monitoring.previousStepSTRING := 'N/A';
   mainPnP.sequence.monitoring.inStepIdle := TRUE;
   mainPnP.sequence.monitoring.inStepStopped := FALSE;
   mainPnP.sequence.monitoring.seqActive := TRUE;
   mainPnP.sequence.monitoring.stepActive := TRUE;
   mainPnP.sequence.monitoring.stepComplete := FALSE;
   mainPnP.sequence.monitoring.executionEnabled := TRUE;
   mainPnP.sequence.monitoring.initRequired := FALSE;
   mainPnP.sequence.monitoring.stepChangeReleased := TRUE;
   mainPnP.sequence.monitoring.justSteppedPulse := FALSE;
   mainPnP.sequence.monitoring.manualControlEnabled := FALSE;
   mainPnP.sequence.monitoring.manualModeChangeEnabled := FALSE;
   mainPnP.sequence.monitoring.memoryStepTimer := 16#0000_4EB7_0DCD_6EA2;
   alignTable.jobs.commands.setJobNumber := 0;
   alignTable.jobs.commands.reset := FALSE;
   alignTable.jobs.status.activeJobNumber := 1;
   alignTable.jobs.status.previousCycleJobNumber := 1;
   alignTable.jobs.status.manualControlEnabled := FALSE;
   alignTable.jobs.status.memoryJobTime := 16#0000_4E8D_4592_AC24;
   alignTable.sequence.commands.setAutomaticMode := FALSE;
   alignTable.sequence.commands.setSingleStepMode := FALSE;
   alignTable.sequence.commands.off := FALSE;
   alignTable.sequence.commands.initialize := FALSE;
   alignTable.sequence.commands.start := FALSE;
   alignTable.sequence.commands.immediateStop := FALSE;
   alignTable.sequence.commands.hold := FALSE;
   alignTable.sequence.commands.nextStep := FALSE;
   alignTable.sequence.commands.interlockStepChange := FALSE;
   alignTable.sequence.monitoring.automaticMode := TRUE;
   alignTable.sequence.monitoring.singleStepMode := FALSE;
   alignTable.sequence.monitoring.currentStep := 160;
   alignTable.sequence.monitoring.nextStep := 160;
   alignTable.sequence.monitoring.previousStep := 142;
   alignTable.sequence.monitoring.currentStepSTRING := 'N/A';
   alignTable.sequence.monitoring.nextStepSTRING := 'N/A';
   alignTable.sequence.monitoring.previousStepSTRING := 'N/A';
   alignTable.sequence.monitoring.inStepIdle := FALSE;
   alignTable.sequence.monitoring.inStepStopped := FALSE;
   alignTable.sequence.monitoring.seqActive := TRUE;
   alignTable.sequence.monitoring.stepActive := TRUE;
   alignTable.sequence.monitoring.stepComplete := FALSE;
   alignTable.sequence.monitoring.executionEnabled := FALSE;
   alignTable.sequence.monitoring.initRequired := FALSE;
   alignTable.sequence.monitoring.stepChangeReleased := TRUE;
   alignTable.sequence.monitoring.justSteppedPulse := FALSE;
   alignTable.sequence.monitoring.manualControlEnabled := FALSE;
   alignTable.sequence.monitoring.manualModeChangeEnabled := FALSE;
   alignTable.sequence.monitoring.memoryStepTimer := 16#0000_4EB6_9139_33B9;
   ngPnP.jobs.commands.setJobNumber := 0;
   ngPnP.jobs.commands.reset := FALSE;
   ngPnP.jobs.status.activeJobNumber := 0;
   ngPnP.jobs.status.previousCycleJobNumber := 0;
   ngPnP.jobs.status.manualControlEnabled := FALSE;
   ngPnP.jobs.status.memoryJobTime := 16#0000_4E8D_4248_232A;
   ngPnP.sequence.commands.setAutomaticMode := FALSE;
   ngPnP.sequence.commands.setSingleStepMode := FALSE;
   ngPnP.sequence.commands.off := FALSE;
   ngPnP.sequence.commands.initialize := FALSE;
   ngPnP.sequence.commands.start := FALSE;
   ngPnP.sequence.commands.immediateStop := FALSE;
   ngPnP.sequence.commands.hold := FALSE;
   ngPnP.sequence.commands.nextStep := FALSE;
   ngPnP.sequence.commands.interlockStepChange := FALSE;
   ngPnP.sequence.monitoring.automaticMode := TRUE;
   ngPnP.sequence.monitoring.singleStepMode := FALSE;
   ngPnP.sequence.monitoring.currentStep := 1;
   ngPnP.sequence.monitoring.nextStep := 1;
   ngPnP.sequence.monitoring.previousStep := 190;
   ngPnP.sequence.monitoring.currentStepSTRING := 'N/A';
   ngPnP.sequence.monitoring.nextStepSTRING := 'N/A';
   ngPnP.sequence.monitoring.previousStepSTRING := 'N/A';
   ngPnP.sequence.monitoring.inStepIdle := TRUE;
   ngPnP.sequence.monitoring.inStepStopped := FALSE;
   ngPnP.sequence.monitoring.seqActive := TRUE;
   ngPnP.sequence.monitoring.stepActive := TRUE;
   ngPnP.sequence.monitoring.stepComplete := FALSE;
   ngPnP.sequence.monitoring.executionEnabled := TRUE;
   ngPnP.sequence.monitoring.initRequired := FALSE;
   ngPnP.sequence.monitoring.stepChangeReleased := TRUE;
   ngPnP.sequence.monitoring.justSteppedPulse := FALSE;
   ngPnP.sequence.monitoring.manualControlEnabled := FALSE;
   ngPnP.sequence.monitoring.manualModeChangeEnabled := FALSE;
   ngPnP.sequence.monitoring.memoryStepTimer := 16#0000_4E8D_4247_6FEB;
   gaugeRnR.jobs.commands.setJobNumber := 0;
   gaugeRnR.jobs.commands.reset := FALSE;
   gaugeRnR.jobs.status.activeJobNumber := 0;
   gaugeRnR.jobs.status.previousCycleJobNumber := 0;
   gaugeRnR.jobs.status.manualControlEnabled := FALSE;
   gaugeRnR.jobs.status.memoryJobTime := 0.0;
   gaugeRnR.sequence.commands.setAutomaticMode := FALSE;
   gaugeRnR.sequence.commands.setSingleStepMode := FALSE;
   gaugeRnR.sequence.commands.off := FALSE;
   gaugeRnR.sequence.commands.initialize := FALSE;
   gaugeRnR.sequence.commands.start := FALSE;
   gaugeRnR.sequence.commands.immediateStop := FALSE;
   gaugeRnR.sequence.commands.hold := FALSE;
   gaugeRnR.sequence.commands.nextStep := FALSE;
   gaugeRnR.sequence.commands.interlockStepChange := FALSE;
   gaugeRnR.sequence.monitoring.automaticMode := TRUE;
   gaugeRnR.sequence.monitoring.singleStepMode := FALSE;
   gaugeRnR.sequence.monitoring.currentStep := 1;
   gaugeRnR.sequence.monitoring.nextStep := 1;
   gaugeRnR.sequence.monitoring.previousStep := 9001;
   gaugeRnR.sequence.monitoring.currentStepSTRING := 'N/A';
   gaugeRnR.sequence.monitoring.nextStepSTRING := 'N/A';
   gaugeRnR.sequence.monitoring.previousStepSTRING := 'N/A';
   gaugeRnR.sequence.monitoring.inStepIdle := TRUE;
   gaugeRnR.sequence.monitoring.inStepStopped := FALSE;
   gaugeRnR.sequence.monitoring.seqActive := TRUE;
   gaugeRnR.sequence.monitoring.stepActive := TRUE;
   gaugeRnR.sequence.monitoring.stepComplete := FALSE;
   gaugeRnR.sequence.monitoring.executionEnabled := TRUE;
   gaugeRnR.sequence.monitoring.initRequired := FALSE;
   gaugeRnR.sequence.monitoring.stepChangeReleased := TRUE;
   gaugeRnR.sequence.monitoring.justSteppedPulse := FALSE;
   gaugeRnR.sequence.monitoring.manualControlEnabled := FALSE;
   gaugeRnR.sequence.monitoring.manualModeChangeEnabled := FALSE;
   gaugeRnR.sequence.monitoring.memoryStepTimer := 16#0000_4E8B_7843_50C0;
   anodeNgCount.referenceDesignator := WSTRING#'Em4 Anode NG Count';
   anodeNgCount.actualCount := 0;
   anodeNgCount.countResetButton := FALSE;
   anodeNgCount.alarmSaveButton := FALSE;
   anodeNgCount.ProcessValue.warningCount := 0;
   anodeNgCount.ProcessValue.faultCount := 0;
   anodeNgCount.SetValue.warningCount := 0;
   anodeNgCount.SetValue.faultCount := 0;
   cmPnp1stAnodeDetect.commands.refreshConfiguration := FALSE;
   cmPnp1stAnodeDetect.commands.editConfiguration := FALSE;
   cmPnp1stAnodeDetect.commands.saveConfiguration := FALSE;
   cmPnp1stAnodeDetect.commands.reset := FALSE;
   cmPnp1stAnodeDetect.monitoring.enable := TRUE;
   cmPnp1stAnodeDetect.monitoring.referenceDesignator := WSTRING#'Pnp1stAnodeDetect';
   cmPnp1stAnodeDetect.monitoring.simulation := FALSE;
   cmPnp1stAnodeDetect.monitoring.processValue := FALSE;
   cmPnp1stAnodeDetect.monitoring.error := FALSE;
   cmPnp1stAnodeDetect.monitoring.status := 16#0000;
   cmPnp1stAnodeDetect.configuration.referenceDesignator := WSTRING#'DigitalSignal';
   cmPnp1stAnodeDetect.configuration.onDelay := T#0MS;
   cmPnp1stAnodeDetect.configuration.offDelay := T#0MS;
   cmPnp1stAnodeDetect.configuration.default := FALSE;
   cmPnp1stAnodeDetect.configuration.invertProcessValue := FALSE;
   cmPnp1stAnodeDetect.configuration.disableAlarms := FALSE;
   cmPnp2ndAnodeDetect.commands.refreshConfiguration := FALSE;
   cmPnp2ndAnodeDetect.commands.editConfiguration := FALSE;
   cmPnp2ndAnodeDetect.commands.saveConfiguration := FALSE;
   cmPnp2ndAnodeDetect.commands.reset := FALSE;
   cmPnp2ndAnodeDetect.monitoring.enable := TRUE;
   cmPnp2ndAnodeDetect.monitoring.referenceDesignator := WSTRING#'Pnp2ndAnodeDetect';
   cmPnp2ndAnodeDetect.monitoring.simulation := FALSE;
   cmPnp2ndAnodeDetect.monitoring.processValue := FALSE;
   cmPnp2ndAnodeDetect.monitoring.error := FALSE;
   cmPnp2ndAnodeDetect.monitoring.status := 16#0000;
   cmPnp2ndAnodeDetect.configuration.referenceDesignator := WSTRING#'DigitalSignal';
   cmPnp2ndAnodeDetect.configuration.onDelay := T#0MS;
   cmPnp2ndAnodeDetect.configuration.offDelay := T#0MS;
   cmPnp2ndAnodeDetect.configuration.default := FALSE;
   cmPnp2ndAnodeDetect.configuration.invertProcessValue := FALSE;
   cmPnp2ndAnodeDetect.configuration.disableAlarms := FALSE;
   cmAnodeAlignTableElectrodeDetect.commands.refreshConfiguration := FALSE;
   cmAnodeAlignTableElectrodeDetect.commands.editConfiguration := FALSE;
   cmAnodeAlignTableElectrodeDetect.commands.saveConfiguration := FALSE;
   cmAnodeAlignTableElectrodeDetect.commands.reset := FALSE;
   cmAnodeAlignTableElectrodeDetect.monitoring.enable := TRUE;
   cmAnodeAlignTableElectrodeDetect.monitoring.referenceDesignator := WSTRING#'AlignTableElectrodeDetect';
   cmAnodeAlignTableElectrodeDetect.monitoring.simulation := FALSE;
   cmAnodeAlignTableElectrodeDetect.monitoring.processValue := FALSE;
   cmAnodeAlignTableElectrodeDetect.monitoring.error := FALSE;
   cmAnodeAlignTableElectrodeDetect.monitoring.status := 16#0000;
   cmAnodeAlignTableElectrodeDetect.configuration.referenceDesignator := WSTRING#'DigitalSignal';
   cmAnodeAlignTableElectrodeDetect.configuration.onDelay := T#0MS;
   cmAnodeAlignTableElectrodeDetect.configuration.offDelay := T#0MS;
   cmAnodeAlignTableElectrodeDetect.configuration.default := FALSE;
   cmAnodeAlignTableElectrodeDetect.configuration.invertProcessValue := FALSE;
   cmAnodeAlignTableElectrodeDetect.configuration.disableAlarms := FALSE;
   cmAnodeNgPnpElectrodeDetect.commands.refreshConfiguration := FALSE;
   cmAnodeNgPnpElectrodeDetect.commands.editConfiguration := FALSE;
   cmAnodeNgPnpElectrodeDetect.commands.saveConfiguration := FALSE;
   cmAnodeNgPnpElectrodeDetect.commands.reset := FALSE;
   cmAnodeNgPnpElectrodeDetect.monitoring.enable := FALSE;
   cmAnodeNgPnpElectrodeDetect.monitoring.referenceDesignator := WSTRING#'';
   cmAnodeNgPnpElectrodeDetect.monitoring.simulation := FALSE;
   cmAnodeNgPnpElectrodeDetect.monitoring.processValue := FALSE;
   cmAnodeNgPnpElectrodeDetect.monitoring.error := FALSE;
   cmAnodeNgPnpElectrodeDetect.monitoring.status := 16#0000;
   cmAnodeNgPnpElectrodeDetect.configuration.referenceDesignator := WSTRING#'DigitalSignal';
   cmAnodeNgPnpElectrodeDetect.configuration.onDelay := T#0MS;
   cmAnodeNgPnpElectrodeDetect.configuration.offDelay := T#0MS;
   cmAnodeNgPnpElectrodeDetect.configuration.default := FALSE;
   cmAnodeNgPnpElectrodeDetect.configuration.invertProcessValue := FALSE;
   cmAnodeNgPnpElectrodeDetect.configuration.disableAlarms := FALSE;
   cmAnodeNgBoxFullSensorDetect.commands.refreshConfiguration := FALSE;
   cmAnodeNgBoxFullSensorDetect.commands.editConfiguration := FALSE;
   cmAnodeNgBoxFullSensorDetect.commands.saveConfiguration := FALSE;
   cmAnodeNgBoxFullSensorDetect.commands.reset := FALSE;
   cmAnodeNgBoxFullSensorDetect.monitoring.enable := TRUE;
   cmAnodeNgBoxFullSensorDetect.monitoring.referenceDesignator := WSTRING#'NgBoxFullSensorDetect';
   cmAnodeNgBoxFullSensorDetect.monitoring.simulation := FALSE;
   cmAnodeNgBoxFullSensorDetect.monitoring.processValue := FALSE;
   cmAnodeNgBoxFullSensorDetect.monitoring.error := FALSE;
   cmAnodeNgBoxFullSensorDetect.monitoring.status := 16#0000;
   cmAnodeNgBoxFullSensorDetect.configuration.referenceDesignator := WSTRING#'DigitalSignal';
   cmAnodeNgBoxFullSensorDetect.configuration.onDelay := T#0MS;
   cmAnodeNgBoxFullSensorDetect.configuration.offDelay := T#0MS;
   cmAnodeNgBoxFullSensorDetect.configuration.default := FALSE;
   cmAnodeNgBoxFullSensorDetect.configuration.invertProcessValue := FALSE;
   cmAnodeNgBoxFullSensorDetect.configuration.disableAlarms := FALSE;
   cmAnodeNgBoxDetect.commands.refreshConfiguration := FALSE;
   cmAnodeNgBoxDetect.commands.editConfiguration := FALSE;
   cmAnodeNgBoxDetect.commands.saveConfiguration := FALSE;
   cmAnodeNgBoxDetect.commands.reset := FALSE;
   cmAnodeNgBoxDetect.monitoring.enable := TRUE;
   cmAnodeNgBoxDetect.monitoring.referenceDesignator := WSTRING#'NgBoxDetect';
   cmAnodeNgBoxDetect.monitoring.simulation := FALSE;
   cmAnodeNgBoxDetect.monitoring.processValue := FALSE;
   cmAnodeNgBoxDetect.monitoring.error := FALSE;
   cmAnodeNgBoxDetect.monitoring.status := 16#0000;
   cmAnodeNgBoxDetect.configuration.referenceDesignator := WSTRING#'DigitalSignal';
   cmAnodeNgBoxDetect.configuration.onDelay := T#0MS;
   cmAnodeNgBoxDetect.configuration.offDelay := T#0MS;
   cmAnodeNgBoxDetect.configuration.default := FALSE;
   cmAnodeNgBoxDetect.configuration.invertProcessValue := FALSE;
   cmAnodeNgBoxDetect.configuration.disableAlarms := FALSE;
   cmAnodeMainPnP1AxisX.commandConfiguration.generalSettings.stopOnError := TRUE;
   cmAnodeMainPnP1AxisX.commandConfiguration.generalSettings.resetWithRestart := FALSE;
   cmAnodeMainPnP1AxisX.commandConfiguration.generalSettings.abortWaitingSyncCmd := TRUE;
   cmAnodeMainPnP1AxisX.commandConfiguration.power.startMode := 1;
   cmAnodeMainPnP1AxisX.commandConfiguration.power.stopMode := 0;
   cmAnodeMainPnP1AxisX.commandConfiguration.power.syncMotionSimulation := FALSE;
   cmAnodeMainPnP1AxisX.commandConfiguration.power.syncMotionSimulationExtendedMode := -1;
   cmAnodeMainPnP1AxisX.commandConfiguration.jog.velocity := 10.0;
   cmAnodeMainPnP1AxisX.commandConfiguration.jog.acceleration := 100.0;
   cmAnodeMainPnP1AxisX.commandConfiguration.jog.deceleration := 100.0;
   cmAnodeMainPnP1AxisX.commandConfiguration.jog.jerk := -1.0;
   cmAnodeMainPnP1AxisX.commandConfiguration.jog.positionControlled := TRUE;
   cmAnodeMainPnP1AxisX.commandConfiguration.jog.increment := 0.0;
   cmAnodeMainPnP1AxisX.commandConfiguration.jog.mode := 0;
   cmAnodeMainPnP1AxisX.commandConfiguration.moveVelocity.velocity := 10.0;
   cmAnodeMainPnP1AxisX.commandConfiguration.moveVelocity.acceleration := 100.0;
   cmAnodeMainPnP1AxisX.commandConfiguration.moveVelocity.deceleration := 100.0;
   cmAnodeMainPnP1AxisX.commandConfiguration.moveVelocity.jerk := -1.0;
   cmAnodeMainPnP1AxisX.commandConfiguration.moveVelocity.direction := 0;
   cmAnodeMainPnP1AxisX.commandConfiguration.moveVelocity.positionControlled := TRUE;
   cmAnodeMainPnP1AxisX.commandConfiguration.moveVelocity.velocityChangeOnTheFly := FALSE;
   cmAnodeMainPnP1AxisX.commandConfiguration.stop.deceleration := -1.0;
   cmAnodeMainPnP1AxisX.commandConfiguration.stop.jerk := -1.0;
   cmAnodeMainPnP1AxisX.commandConfiguration.stop.abortAcceleration := FALSE;
   cmAnodeMainPnP1AxisX.commandConfiguration.fastStop.deceleration := -1.0;
   cmAnodeMainPnP1AxisX.commandConfiguration.fastStop.jerk := -1.0;
   cmAnodeMainPnP1AxisX.commandConfiguration.fastStop.abortAcceleration := FALSE;
   cmAnodeMainPnP1AxisX.commandConfiguration.fastStop.replaceStopPossible := FALSE;
   cmAnodeMainPnP1AxisX.commandConfiguration.torqueLimiting.limit := -1.0;
   cmAnodeMainPnP1AxisX.commandConfiguration.torqueLimiting.mode := 0;
   cmAnodeMainPnP1AxisX.commandConfiguration.homing.position := 0.0;
   cmAnodeMainPnP1AxisX.commandConfiguration.homing.mode := 0;
   cmAnodeMainPnP1AxisX.commandConfiguration.homing.sensor := 0;
   cmAnodeMainPnP1AxisX.commandConfiguration.homing.extendedMode := -1;
   cmAnodeMainPnP1AxisX.commandConfiguration.homing.extendedModeTorqueLimit := 0.0;
   cmAnodeMainPnP1AxisX.commandConfiguration.homing.extendedModeTargetPosition := 0.0;
   cmAnodeMainPnP1AxisX.commandConfiguration.posRelative.distance := 0.0;
   cmAnodeMainPnP1AxisX.commandConfiguration.posRelative.velocity := 10.0;
   cmAnodeMainPnP1AxisX.commandConfiguration.posRelative.acceleration := 100.0;
   cmAnodeMainPnP1AxisX.commandConfiguration.posRelative.deceleration := 100.0;
   cmAnodeMainPnP1AxisX.commandConfiguration.posRelative.jerk := -1.0;
   cmAnodeMainPnP1AxisX.commandConfiguration.posRelative.direction := 0;
   cmAnodeMainPnP1AxisX.commandConfiguration.posAbsolute.position := 0.0;
   cmAnodeMainPnP1AxisX.commandConfiguration.posAbsolute.velocity := -1.0;
   cmAnodeMainPnP1AxisX.commandConfiguration.posAbsolute.acceleration := -1.0;
   cmAnodeMainPnP1AxisX.commandConfiguration.posAbsolute.deceleration := -1.0;
   cmAnodeMainPnP1AxisX.commandConfiguration.posAbsolute.jerk := -1.0;
   cmAnodeMainPnP1AxisX.commandConfiguration.posAbsolute.direction := 1;
   cmAnodeMainPnP1AxisX.commandConfiguration.posAbsolute.positionChangeOnTheFly := FALSE;
   cmAnodeMainPnP1AxisX.commandConfiguration.posAbsolute.velocityChangeOnTheFly := FALSE;
   cmAnodeMainPnP1AxisX.commandConfiguration.posSuperimposed.distance := 0.0;
   cmAnodeMainPnP1AxisX.commandConfiguration.posSuperimposed.velocityDiff := -1.0;
   cmAnodeMainPnP1AxisX.commandConfiguration.posSuperimposed.acceleration := -1.0;
   cmAnodeMainPnP1AxisX.commandConfiguration.posSuperimposed.deceleration := -1.0;
   cmAnodeMainPnP1AxisX.commandConfiguration.posSuperimposed.jerk := -1.0;
   cmAnodeMainPnP1AxisX.commandConfiguration.posSuperimposed.direction := 0;
   cmAnodeMainPnP1AxisX.commandConfiguration.haltSuperimposed.deceleration := -1.0;
   cmAnodeMainPnP1AxisX.commandConfiguration.haltSuperimposed.jerk := -1.0;
   cmAnodeMainPnP1AxisX.commandConfiguration.haltSuperimposed.abortAcceleration := FALSE;
   cmAnodeMainPnP1AxisX.commandConfiguration.gearInRelative.ratioNumerator := 1;
   cmAnodeMainPnP1AxisX.commandConfiguration.gearInRelative.ratioDenominator := 1;
   cmAnodeMainPnP1AxisX.commandConfiguration.gearInRelative.acceleration := -1.0;
   cmAnodeMainPnP1AxisX.commandConfiguration.gearInRelative.deceleration := -1.0;
   cmAnodeMainPnP1AxisX.commandConfiguration.gearInRelative.jerk := -1.0;
   cmAnodeMainPnP1AxisX.commandConfiguration.gearInRelative.ratioChangeOnTheFly := FALSE;
   cmAnodeMainPnP1AxisX.commandConfiguration.gearInAbsolute.ratioNumerator := 1;
   cmAnodeMainPnP1AxisX.commandConfiguration.gearInAbsolute.ratioDenominator := 1;
   cmAnodeMainPnP1AxisX.commandConfiguration.gearInAbsolute.masterSyncPosition := 0.0;
   cmAnodeMainPnP1AxisX.commandConfiguration.gearInAbsolute.slaveSyncPosition := 0.0;
   cmAnodeMainPnP1AxisX.commandConfiguration.gearInAbsolute.syncProfileReference := 1;
   cmAnodeMainPnP1AxisX.commandConfiguration.gearInAbsolute.masterStartDistance := 0.0;
   cmAnodeMainPnP1AxisX.commandConfiguration.gearInAbsolute.velocity := -1.0;
   cmAnodeMainPnP1AxisX.commandConfiguration.gearInAbsolute.acceleration := -1.0;
   cmAnodeMainPnP1AxisX.commandConfiguration.gearInAbsolute.deceleration := -1.0;
   cmAnodeMainPnP1AxisX.commandConfiguration.gearInAbsolute.jerk := -1.0;
   cmAnodeMainPnP1AxisX.commandConfiguration.gearInAbsolute.syncDirection := 1;
   cmAnodeMainPnP1AxisX.commandConfiguration.gearInAbsolute.ratioChangeOnTheFly := FALSE;
   cmAnodeMainPnP1AxisX.commandConfiguration.gearInVelocity.continuousUpdate := FALSE;
   cmAnodeMainPnP1AxisX.commandConfiguration.gearInVelocity.ratioNumerator := 1;
   cmAnodeMainPnP1AxisX.commandConfiguration.gearInVelocity.ratioDenominator := 1;
   cmAnodeMainPnP1AxisX.commandConfiguration.gearInVelocity.acceleration := -1.0;
   cmAnodeMainPnP1AxisX.commandConfiguration.gearInVelocity.deceleration := -1.0;
   cmAnodeMainPnP1AxisX.commandConfiguration.gearInVelocity.jerk := -1.0;
   cmAnodeMainPnP1AxisX.commandConfiguration.gearInVelocity.positionControlled := FALSE;
   cmAnodeMainPnP1AxisX.commandConfiguration.camIn.masterOffset := 0.0;
   cmAnodeMainPnP1AxisX.commandConfiguration.camIn.slaveOffset := 0.0;
   cmAnodeMainPnP1AxisX.commandConfiguration.camIn.masterScaling := 1.0;
   cmAnodeMainPnP1AxisX.commandConfiguration.camIn.slaveScaling := 1.0;
   cmAnodeMainPnP1AxisX.commandConfiguration.camIn.masterSyncPosition := 0.0;
   cmAnodeMainPnP1AxisX.commandConfiguration.camIn.syncProfileReference := 1;
   cmAnodeMainPnP1AxisX.commandConfiguration.camIn.masterStartDistance := 0.0;
   cmAnodeMainPnP1AxisX.commandConfiguration.camIn.velocity := -1.0;
   cmAnodeMainPnP1AxisX.commandConfiguration.camIn.acceleration := -1.0;
   cmAnodeMainPnP1AxisX.commandConfiguration.camIn.deceleration := -1.0;
   cmAnodeMainPnP1AxisX.commandConfiguration.camIn.jerk := -1.0;
   cmAnodeMainPnP1AxisX.commandConfiguration.camIn.applicationMode := 0;
   cmAnodeMainPnP1AxisX.commandConfiguration.camIn.syncDirection := 1;
   cmAnodeMainPnP1AxisX.commandConfiguration.gearOutCamOut.slavePosition := 0.0;
   cmAnodeMainPnP1AxisX.commandConfiguration.gearOutCamOut.syncProfileReference := 1;
   cmAnodeMainPnP1AxisX.commandConfiguration.gearOutCamOut.masterStopDistance := 0.0;
   cmAnodeMainPnP1AxisX.commandConfiguration.gearOutCamOut.deceleration := -1.0;
   cmAnodeMainPnP1AxisX.commandConfiguration.gearOutCamOut.jerk := -1.0;
   cmAnodeMainPnP1AxisX.commandConfiguration.gearOutCamOut.syncOutDirection := 3;
   cmAnodeMainPnP1AxisX.commandConfiguration.gearOutCamOut.gearOutCamOutMode := -1;
   cmAnodeMainPnP1AxisX.commandConfiguration.phasing.phaseShift := 0.0;
   cmAnodeMainPnP1AxisX.commandConfiguration.phasing.velocity := -1.0;
   cmAnodeMainPnP1AxisX.commandConfiguration.phasing.acceleration := -1.0;
   cmAnodeMainPnP1AxisX.commandConfiguration.phasing.deceleration := -1.0;
   cmAnodeMainPnP1AxisX.commandConfiguration.phasing.jerk := -1.0;
   cmAnodeMainPnP1AxisX.commandConfiguration.phasing.profileReference := 0;
   cmAnodeMainPnP1AxisX.commandConfiguration.phasing.phasingDistance := 0.0;
   cmAnodeMainPnP1AxisX.commandConfiguration.phasing.startPosition := 0.0;
   cmAnodeMainPnP1AxisX.commandConfiguration.phasing.direction := 3;
   cmAnodeMainPnP1AxisX.commandConfiguration.phasing.phaseAbsolute := TRUE;
   cmAnodeMainPnP1AxisX.commandConfiguration.phasing.phaseShiftChangeOnTheFly := FALSE;
   cmAnodeMainPnP1AxisX.commandConfiguration.offset.offset := 0.0;
   cmAnodeMainPnP1AxisX.commandConfiguration.offset.profileReference := 1;
   cmAnodeMainPnP1AxisX.commandConfiguration.offset.offsetDistance := 0.0;
   cmAnodeMainPnP1AxisX.commandConfiguration.offset.startPosition := 0.0;
   cmAnodeMainPnP1AxisX.commandConfiguration.offset.direction := 3;
   cmAnodeMainPnP1AxisX.commandConfiguration.offset.offsetAbsolute := TRUE;
   cmAnodeMainPnP1AxisX.commandConfiguration.offset.offsetChangeOnTheFly := FALSE;
   cmAnodeMainPnP1AxisX.commands.enableMasterControl := TRUE;
   cmAnodeMainPnP1AxisX.commands.enableAxis := FALSE;
   cmAnodeMainPnP1AxisX.commands.resetAxis := FALSE;
   cmAnodeMainPnP1AxisX.commands.openBrake := FALSE;
   cmAnodeMainPnP1AxisX.commands.jogForward := FALSE;
   cmAnodeMainPnP1AxisX.commands.jogBackward := FALSE;
   cmAnodeMainPnP1AxisX.commands.moveVelocity := FALSE;
   cmAnodeMainPnP1AxisX.commands.stop := FALSE;
   cmAnodeMainPnP1AxisX.commands.fastStop := FALSE;
   cmAnodeMainPnP1AxisX.commands.torqueLimiting := FALSE;
   cmAnodeMainPnP1AxisX.commands.homing := FALSE;
   cmAnodeMainPnP1AxisX.commands.posRelative := FALSE;
   cmAnodeMainPnP1AxisX.commands.posAbsolute := FALSE;
   cmAnodeMainPnP1AxisX.commands.posSuperimposed := FALSE;
   cmAnodeMainPnP1AxisX.commands.haltSuperimposed := FALSE;
   cmAnodeMainPnP1AxisX.commands.selectSetPosition := 1;
   cmAnodeMainPnP1AxisX.commands.uploadParameters := FALSE;
   cmAnodeMainPnP1AxisX.commands.refreshConfiguration := FALSE;
   cmAnodeMainPnP1AxisX.commands.editConfiguration := FALSE;
   cmAnodeMainPnP1AxisX.commands.saveConfiguration := FALSE;
   cmAnodeMainPnP1AxisX.commands.uploadCurrentTorque := FALSE;
   cmAnodeMainPnP1AxisX.commands.reset := FALSE;
   cmAnodeMainPnP1AxisX.monitoring.enable := TRUE;
   cmAnodeMainPnP1AxisX.monitoring.referenceDesignator := WSTRING#'AnodeMainPnP1AxisX';
   cmAnodeMainPnP1AxisX.monitoring.enabled := TRUE;
   cmAnodeMainPnP1AxisX.monitoring.enableManualCmds := FALSE;
   cmAnodeMainPnP1AxisX.monitoring.reset := FALSE;
   cmAnodeMainPnP1AxisX.monitoring.resetAxis := FALSE;
   cmAnodeMainPnP1AxisX.monitoring.enableAxis := TRUE;
   cmAnodeMainPnP1AxisX.monitoring.openBrake := FALSE;
   cmAnodeMainPnP1AxisX.monitoring.jogBackward := FALSE;
   cmAnodeMainPnP1AxisX.monitoring.jogForward := FALSE;
   cmAnodeMainPnP1AxisX.monitoring.moveVelocity := FALSE;
   cmAnodeMainPnP1AxisX.monitoring.stop := FALSE;
   cmAnodeMainPnP1AxisX.monitoring.fastStop := FALSE;
   cmAnodeMainPnP1AxisX.monitoring.torqueLimiting := FALSE;
   cmAnodeMainPnP1AxisX.monitoring.homing := FALSE;
   cmAnodeMainPnP1AxisX.monitoring.posRelative := FALSE;
   cmAnodeMainPnP1AxisX.monitoring.posAbsolute := FALSE;
   cmAnodeMainPnP1AxisX.monitoring.posSuperimposed := FALSE;
   cmAnodeMainPnP1AxisX.monitoring.haltSuperimposed := FALSE;
   cmAnodeMainPnP1AxisX.monitoring.brakeOpened := FALSE;
   cmAnodeMainPnP1AxisX.monitoring.axisEnabled := TRUE;
   cmAnodeMainPnP1AxisX.monitoring.resetActive := FALSE;
   cmAnodeMainPnP1AxisX.monitoring.inVelocity := FALSE;
   cmAnodeMainPnP1AxisX.monitoring.inLimitation := FALSE;
   cmAnodeMainPnP1AxisX.monitoring.inClamping := FALSE;
   cmAnodeMainPnP1AxisX.monitoring.startSync := FALSE;
   cmAnodeMainPnP1AxisX.monitoring.inSync := FALSE;
   cmAnodeMainPnP1AxisX.monitoring.inSimulation := FALSE;
   cmAnodeMainPnP1AxisX.monitoring.jogSelected := FALSE;
   cmAnodeMainPnP1AxisX.monitoring.moveVelocitySelected := FALSE;
   cmAnodeMainPnP1AxisX.monitoring.stopSelected := FALSE;
   cmAnodeMainPnP1AxisX.monitoring.fastStopSelected := FALSE;
   cmAnodeMainPnP1AxisX.monitoring.torqueLimitingSelected := FALSE;
   cmAnodeMainPnP1AxisX.monitoring.homingSelected := FALSE;
   cmAnodeMainPnP1AxisX.monitoring.posRelativeSelected := FALSE;
   cmAnodeMainPnP1AxisX.monitoring.posAbsoluteSelected := FALSE;
   cmAnodeMainPnP1AxisX.monitoring.posSuperimposedSelected := FALSE;
   cmAnodeMainPnP1AxisX.monitoring.haltSuperimposedSelected := FALSE;
   cmAnodeMainPnP1AxisX.monitoring.commandBusy := FALSE;
   cmAnodeMainPnP1AxisX.monitoring.commandDone := FALSE;
   cmAnodeMainPnP1AxisX.monitoring.commandAborted := FALSE;
   cmAnodeMainPnP1AxisX.monitoring.homingCommandBusy := FALSE;
   cmAnodeMainPnP1AxisX.monitoring.homingCommandDone := FALSE;
   cmAnodeMainPnP1AxisX.monitoring.homingCommandAborted := FALSE;
   cmAnodeMainPnP1AxisX.monitoring.superimposedBusy := FALSE;
   cmAnodeMainPnP1AxisX.monitoring.superimposedDone := FALSE;
   cmAnodeMainPnP1AxisX.monitoring.superimposedAborted := FALSE;
   cmAnodeMainPnP1AxisX.monitoring.selectSetPosition := 1;
   cmAnodeMainPnP1AxisX.monitoring.selectionController := FALSE;
   cmAnodeMainPnP1AxisX.monitoring.interlockGeneral := TRUE;
   cmAnodeMainPnP1AxisX.monitoring.interlockJogForward := TRUE;
   cmAnodeMainPnP1AxisX.monitoring.interlockJogBackward := TRUE;
   cmAnodeMainPnP1AxisX.monitoring.interlockWarningGeneral := FALSE;
   cmAnodeMainPnP1AxisX.monitoring.interlockWarningJogForward := FALSE;
   cmAnodeMainPnP1AxisX.monitoring.interlockWarningJogBackward := FALSE;
   cmAnodeMainPnP1AxisX.monitoring.valid := TRUE;
   cmAnodeMainPnP1AxisX.monitoring.busy := TRUE;
   cmAnodeMainPnP1AxisX.monitoring.error := FALSE;
   cmAnodeMainPnP1AxisX.monitoring.status := 16#7002;
   cmAnodeMainPnP1AxisX.monitoring.subfunctionStatus := 16#0000;
   cmAnodeMainPnP1AxisX.monitoring.actualPosition := 539.98;
   cmAnodeMainPnP1AxisX.monitoring.actualSpeed := 6.62553364956176;
   cmAnodeMainPnP1AxisX.monitoring.speedUnit := 1062;
   cmAnodeMainPnP1AxisX.monitoring.positionUnit := 1013;
   cmAnodeMainPnP1AxisX.monitoring.axisStatus1 := 16#0240_4021;
   cmAnodeMainPnP1AxisX.monitoring.axisStatus2 := 16#0000_0000;
   cmAnodeMainPnP1AxisX.monitoring.axisType := 1;
   cmAnodeMainPnP1AxisX.monitoring.maxVelocity := 2500.0;
   cmAnodeMainPnP1AxisX.monitoring.actualCurrent := 0.0;
   cmAnodeMainPnP1AxisX.monitoring.actualTorque := 0.0;
   cmAnodeMainPnP1AxisX.monitoring.velocityOverrideEnabled := FALSE;
   cmAnodeMainPnP1AxisX.monitoring.sinaParaError := FALSE;
   cmAnodeMainPnP1AxisX.monitoring.sinaParaStatus := 16#0000_0000;
   cmAnodeMainPnP1AxisX.configuration.referenceDesignator := WSTRING#'AnodeMainPnP1AxisX';
   cmAnodeMainPnP1AxisX.configuration.disableAlarms := FALSE;
   cmAnodeMainPnP1AxisX.configuration.masterControlPopUp := TRUE;
   cmAnodeMainPnP1AxisX.configuration.setPositions[0].position := 540.0;
   cmAnodeMainPnP1AxisX.configuration.setPositions[1].position := 0.0;
   cmAnodeMainPnP1AxisX.configuration.setPositions[2].position := -5.0;
   cmAnodeMainPnP1AxisX.configuration.setPositions[3..15].position := 0.0;
   cmAnodeMainPnP1AxisX.configuration.setPositions[0..1].velocity := 500.0;
   cmAnodeMainPnP1AxisX.configuration.setPositions[2].velocity := 100.0;
   cmAnodeMainPnP1AxisX.configuration.setPositions[3..15].velocity := -1.0;
   cmAnodeMainPnP1AxisX.configuration.setPositions[0..1].acceleration := 5000.0;
   cmAnodeMainPnP1AxisX.configuration.setPositions[2].acceleration := 30.0;
   cmAnodeMainPnP1AxisX.configuration.setPositions[3..15].acceleration := -1.0;
   cmAnodeMainPnP1AxisX.configuration.setPositions[0..1].deceleration := 5000.0;
   cmAnodeMainPnP1AxisX.configuration.setPositions[2].deceleration := 30.0;
   cmAnodeMainPnP1AxisX.configuration.setPositions[3..15].deceleration := -1.0;
   cmAnodeMainPnP1AxisX.configuration.setPositions[0..15]."name" := '';
   cmAnodeMainPnP2AxisX.commandConfiguration.generalSettings.stopOnError := TRUE;
   cmAnodeMainPnP2AxisX.commandConfiguration.generalSettings.resetWithRestart := FALSE;
   cmAnodeMainPnP2AxisX.commandConfiguration.generalSettings.abortWaitingSyncCmd := TRUE;
   cmAnodeMainPnP2AxisX.commandConfiguration.power.startMode := 1;
   cmAnodeMainPnP2AxisX.commandConfiguration.power.stopMode := 0;
   cmAnodeMainPnP2AxisX.commandConfiguration.power.syncMotionSimulation := FALSE;
   cmAnodeMainPnP2AxisX.commandConfiguration.power.syncMotionSimulationExtendedMode := -1;
   cmAnodeMainPnP2AxisX.commandConfiguration.jog.velocity := 10.0;
   cmAnodeMainPnP2AxisX.commandConfiguration.jog.acceleration := 100.0;
   cmAnodeMainPnP2AxisX.commandConfiguration.jog.deceleration := 100.0;
   cmAnodeMainPnP2AxisX.commandConfiguration.jog.jerk := -1.0;
   cmAnodeMainPnP2AxisX.commandConfiguration.jog.positionControlled := TRUE;
   cmAnodeMainPnP2AxisX.commandConfiguration.jog.increment := 0.0;
   cmAnodeMainPnP2AxisX.commandConfiguration.jog.mode := 0;
   cmAnodeMainPnP2AxisX.commandConfiguration.moveVelocity.velocity := 10.0;
   cmAnodeMainPnP2AxisX.commandConfiguration.moveVelocity.acceleration := 100.0;
   cmAnodeMainPnP2AxisX.commandConfiguration.moveVelocity.deceleration := 100.0;
   cmAnodeMainPnP2AxisX.commandConfiguration.moveVelocity.jerk := -1.0;
   cmAnodeMainPnP2AxisX.commandConfiguration.moveVelocity.direction := 0;
   cmAnodeMainPnP2AxisX.commandConfiguration.moveVelocity.positionControlled := TRUE;
   cmAnodeMainPnP2AxisX.commandConfiguration.moveVelocity.velocityChangeOnTheFly := FALSE;
   cmAnodeMainPnP2AxisX.commandConfiguration.stop.deceleration := -1.0;
   cmAnodeMainPnP2AxisX.commandConfiguration.stop.jerk := -1.0;
   cmAnodeMainPnP2AxisX.commandConfiguration.stop.abortAcceleration := FALSE;
   cmAnodeMainPnP2AxisX.commandConfiguration.fastStop.deceleration := -1.0;
   cmAnodeMainPnP2AxisX.commandConfiguration.fastStop.jerk := -1.0;
   cmAnodeMainPnP2AxisX.commandConfiguration.fastStop.abortAcceleration := FALSE;
   cmAnodeMainPnP2AxisX.commandConfiguration.fastStop.replaceStopPossible := FALSE;
   cmAnodeMainPnP2AxisX.commandConfiguration.torqueLimiting.limit := -1.0;
   cmAnodeMainPnP2AxisX.commandConfiguration.torqueLimiting.mode := 0;
   cmAnodeMainPnP2AxisX.commandConfiguration.homing.position := 0.0;
   cmAnodeMainPnP2AxisX.commandConfiguration.homing.mode := 0;
   cmAnodeMainPnP2AxisX.commandConfiguration.homing.sensor := 0;
   cmAnodeMainPnP2AxisX.commandConfiguration.homing.extendedMode := -1;
   cmAnodeMainPnP2AxisX.commandConfiguration.homing.extendedModeTorqueLimit := 0.0;
   cmAnodeMainPnP2AxisX.commandConfiguration.homing.extendedModeTargetPosition := 0.0;
   cmAnodeMainPnP2AxisX.commandConfiguration.posRelative.distance := 0.0;
   cmAnodeMainPnP2AxisX.commandConfiguration.posRelative.velocity := 10.0;
   cmAnodeMainPnP2AxisX.commandConfiguration.posRelative.acceleration := 100.0;
   cmAnodeMainPnP2AxisX.commandConfiguration.posRelative.deceleration := 100.0;
   cmAnodeMainPnP2AxisX.commandConfiguration.posRelative.jerk := -1.0;
   cmAnodeMainPnP2AxisX.commandConfiguration.posRelative.direction := 0;
   cmAnodeMainPnP2AxisX.commandConfiguration.posAbsolute.position := 0.0;
   cmAnodeMainPnP2AxisX.commandConfiguration.posAbsolute.velocity := -1.0;
   cmAnodeMainPnP2AxisX.commandConfiguration.posAbsolute.acceleration := -1.0;
   cmAnodeMainPnP2AxisX.commandConfiguration.posAbsolute.deceleration := -1.0;
   cmAnodeMainPnP2AxisX.commandConfiguration.posAbsolute.jerk := -1.0;
   cmAnodeMainPnP2AxisX.commandConfiguration.posAbsolute.direction := 1;
   cmAnodeMainPnP2AxisX.commandConfiguration.posAbsolute.positionChangeOnTheFly := FALSE;
   cmAnodeMainPnP2AxisX.commandConfiguration.posAbsolute.velocityChangeOnTheFly := FALSE;
   cmAnodeMainPnP2AxisX.commandConfiguration.posSuperimposed.distance := 0.0;
   cmAnodeMainPnP2AxisX.commandConfiguration.posSuperimposed.velocityDiff := -1.0;
   cmAnodeMainPnP2AxisX.commandConfiguration.posSuperimposed.acceleration := -1.0;
   cmAnodeMainPnP2AxisX.commandConfiguration.posSuperimposed.deceleration := -1.0;
   cmAnodeMainPnP2AxisX.commandConfiguration.posSuperimposed.jerk := -1.0;
   cmAnodeMainPnP2AxisX.commandConfiguration.posSuperimposed.direction := 0;
   cmAnodeMainPnP2AxisX.commandConfiguration.haltSuperimposed.deceleration := -1.0;
   cmAnodeMainPnP2AxisX.commandConfiguration.haltSuperimposed.jerk := -1.0;
   cmAnodeMainPnP2AxisX.commandConfiguration.haltSuperimposed.abortAcceleration := FALSE;
   cmAnodeMainPnP2AxisX.commandConfiguration.gearInRelative.ratioNumerator := 1;
   cmAnodeMainPnP2AxisX.commandConfiguration.gearInRelative.ratioDenominator := 1;
   cmAnodeMainPnP2AxisX.commandConfiguration.gearInRelative.acceleration := -1.0;
   cmAnodeMainPnP2AxisX.commandConfiguration.gearInRelative.deceleration := -1.0;
   cmAnodeMainPnP2AxisX.commandConfiguration.gearInRelative.jerk := -1.0;
   cmAnodeMainPnP2AxisX.commandConfiguration.gearInRelative.ratioChangeOnTheFly := FALSE;
   cmAnodeMainPnP2AxisX.commandConfiguration.gearInAbsolute.ratioNumerator := 1;
   cmAnodeMainPnP2AxisX.commandConfiguration.gearInAbsolute.ratioDenominator := 1;
   cmAnodeMainPnP2AxisX.commandConfiguration.gearInAbsolute.masterSyncPosition := 0.0;
   cmAnodeMainPnP2AxisX.commandConfiguration.gearInAbsolute.slaveSyncPosition := 0.0;
   cmAnodeMainPnP2AxisX.commandConfiguration.gearInAbsolute.syncProfileReference := 1;
   cmAnodeMainPnP2AxisX.commandConfiguration.gearInAbsolute.masterStartDistance := 0.0;
   cmAnodeMainPnP2AxisX.commandConfiguration.gearInAbsolute.velocity := -1.0;
   cmAnodeMainPnP2AxisX.commandConfiguration.gearInAbsolute.acceleration := -1.0;
   cmAnodeMainPnP2AxisX.commandConfiguration.gearInAbsolute.deceleration := -1.0;
   cmAnodeMainPnP2AxisX.commandConfiguration.gearInAbsolute.jerk := -1.0;
   cmAnodeMainPnP2AxisX.commandConfiguration.gearInAbsolute.syncDirection := 1;
   cmAnodeMainPnP2AxisX.commandConfiguration.gearInAbsolute.ratioChangeOnTheFly := FALSE;
   cmAnodeMainPnP2AxisX.commandConfiguration.gearInVelocity.continuousUpdate := FALSE;
   cmAnodeMainPnP2AxisX.commandConfiguration.gearInVelocity.ratioNumerator := 1;
   cmAnodeMainPnP2AxisX.commandConfiguration.gearInVelocity.ratioDenominator := 1;
   cmAnodeMainPnP2AxisX.commandConfiguration.gearInVelocity.acceleration := -1.0;
   cmAnodeMainPnP2AxisX.commandConfiguration.gearInVelocity.deceleration := -1.0;
   cmAnodeMainPnP2AxisX.commandConfiguration.gearInVelocity.jerk := -1.0;
   cmAnodeMainPnP2AxisX.commandConfiguration.gearInVelocity.positionControlled := FALSE;
   cmAnodeMainPnP2AxisX.commandConfiguration.camIn.masterOffset := 0.0;
   cmAnodeMainPnP2AxisX.commandConfiguration.camIn.slaveOffset := 0.0;
   cmAnodeMainPnP2AxisX.commandConfiguration.camIn.masterScaling := 1.0;
   cmAnodeMainPnP2AxisX.commandConfiguration.camIn.slaveScaling := 1.0;
   cmAnodeMainPnP2AxisX.commandConfiguration.camIn.masterSyncPosition := 0.0;
   cmAnodeMainPnP2AxisX.commandConfiguration.camIn.syncProfileReference := 1;
   cmAnodeMainPnP2AxisX.commandConfiguration.camIn.masterStartDistance := 0.0;
   cmAnodeMainPnP2AxisX.commandConfiguration.camIn.velocity := -1.0;
   cmAnodeMainPnP2AxisX.commandConfiguration.camIn.acceleration := -1.0;
   cmAnodeMainPnP2AxisX.commandConfiguration.camIn.deceleration := -1.0;
   cmAnodeMainPnP2AxisX.commandConfiguration.camIn.jerk := -1.0;
   cmAnodeMainPnP2AxisX.commandConfiguration.camIn.applicationMode := 0;
   cmAnodeMainPnP2AxisX.commandConfiguration.camIn.syncDirection := 1;
   cmAnodeMainPnP2AxisX.commandConfiguration.gearOutCamOut.slavePosition := 0.0;
   cmAnodeMainPnP2AxisX.commandConfiguration.gearOutCamOut.syncProfileReference := 1;
   cmAnodeMainPnP2AxisX.commandConfiguration.gearOutCamOut.masterStopDistance := 0.0;
   cmAnodeMainPnP2AxisX.commandConfiguration.gearOutCamOut.deceleration := -1.0;
   cmAnodeMainPnP2AxisX.commandConfiguration.gearOutCamOut.jerk := -1.0;
   cmAnodeMainPnP2AxisX.commandConfiguration.gearOutCamOut.syncOutDirection := 3;
   cmAnodeMainPnP2AxisX.commandConfiguration.gearOutCamOut.gearOutCamOutMode := -1;
   cmAnodeMainPnP2AxisX.commandConfiguration.phasing.phaseShift := 0.0;
   cmAnodeMainPnP2AxisX.commandConfiguration.phasing.velocity := -1.0;
   cmAnodeMainPnP2AxisX.commandConfiguration.phasing.acceleration := -1.0;
   cmAnodeMainPnP2AxisX.commandConfiguration.phasing.deceleration := -1.0;
   cmAnodeMainPnP2AxisX.commandConfiguration.phasing.jerk := -1.0;
   cmAnodeMainPnP2AxisX.commandConfiguration.phasing.profileReference := 0;
   cmAnodeMainPnP2AxisX.commandConfiguration.phasing.phasingDistance := 0.0;
   cmAnodeMainPnP2AxisX.commandConfiguration.phasing.startPosition := 0.0;
   cmAnodeMainPnP2AxisX.commandConfiguration.phasing.direction := 3;
   cmAnodeMainPnP2AxisX.commandConfiguration.phasing.phaseAbsolute := TRUE;
   cmAnodeMainPnP2AxisX.commandConfiguration.phasing.phaseShiftChangeOnTheFly := FALSE;
   cmAnodeMainPnP2AxisX.commandConfiguration.offset.offset := 0.0;
   cmAnodeMainPnP2AxisX.commandConfiguration.offset.profileReference := 1;
   cmAnodeMainPnP2AxisX.commandConfiguration.offset.offsetDistance := 0.0;
   cmAnodeMainPnP2AxisX.commandConfiguration.offset.startPosition := 0.0;
   cmAnodeMainPnP2AxisX.commandConfiguration.offset.direction := 3;
   cmAnodeMainPnP2AxisX.commandConfiguration.offset.offsetAbsolute := TRUE;
   cmAnodeMainPnP2AxisX.commandConfiguration.offset.offsetChangeOnTheFly := FALSE;
   cmAnodeMainPnP2AxisX.commands.enableMasterControl := TRUE;
   cmAnodeMainPnP2AxisX.commands.enableAxis := FALSE;
   cmAnodeMainPnP2AxisX.commands.resetAxis := FALSE;
   cmAnodeMainPnP2AxisX.commands.openBrake := FALSE;
   cmAnodeMainPnP2AxisX.commands.jogForward := FALSE;
   cmAnodeMainPnP2AxisX.commands.jogBackward := FALSE;
   cmAnodeMainPnP2AxisX.commands.moveVelocity := FALSE;
   cmAnodeMainPnP2AxisX.commands.stop := FALSE;
   cmAnodeMainPnP2AxisX.commands.fastStop := FALSE;
   cmAnodeMainPnP2AxisX.commands.torqueLimiting := FALSE;
   cmAnodeMainPnP2AxisX.commands.homing := FALSE;
   cmAnodeMainPnP2AxisX.commands.posRelative := FALSE;
   cmAnodeMainPnP2AxisX.commands.posAbsolute := FALSE;
   cmAnodeMainPnP2AxisX.commands.posSuperimposed := FALSE;
   cmAnodeMainPnP2AxisX.commands.haltSuperimposed := FALSE;
   cmAnodeMainPnP2AxisX.commands.selectSetPosition := 1;
   cmAnodeMainPnP2AxisX.commands.uploadParameters := FALSE;
   cmAnodeMainPnP2AxisX.commands.refreshConfiguration := FALSE;
   cmAnodeMainPnP2AxisX.commands.editConfiguration := FALSE;
   cmAnodeMainPnP2AxisX.commands.saveConfiguration := FALSE;
   cmAnodeMainPnP2AxisX.commands.uploadCurrentTorque := FALSE;
   cmAnodeMainPnP2AxisX.commands.reset := FALSE;
   cmAnodeMainPnP2AxisX.monitoring.enable := TRUE;
   cmAnodeMainPnP2AxisX.monitoring.referenceDesignator := WSTRING#'AnodeMainPnP2AxisX';
   cmAnodeMainPnP2AxisX.monitoring.enabled := TRUE;
   cmAnodeMainPnP2AxisX.monitoring.enableManualCmds := FALSE;
   cmAnodeMainPnP2AxisX.monitoring.reset := FALSE;
   cmAnodeMainPnP2AxisX.monitoring.resetAxis := FALSE;
   cmAnodeMainPnP2AxisX.monitoring.enableAxis := TRUE;
   cmAnodeMainPnP2AxisX.monitoring.openBrake := FALSE;
   cmAnodeMainPnP2AxisX.monitoring.jogBackward := FALSE;
   cmAnodeMainPnP2AxisX.monitoring.jogForward := FALSE;
   cmAnodeMainPnP2AxisX.monitoring.moveVelocity := FALSE;
   cmAnodeMainPnP2AxisX.monitoring.stop := FALSE;
   cmAnodeMainPnP2AxisX.monitoring.fastStop := FALSE;
   cmAnodeMainPnP2AxisX.monitoring.torqueLimiting := FALSE;
   cmAnodeMainPnP2AxisX.monitoring.homing := FALSE;
   cmAnodeMainPnP2AxisX.monitoring.posRelative := FALSE;
   cmAnodeMainPnP2AxisX.monitoring.posAbsolute := FALSE;
   cmAnodeMainPnP2AxisX.monitoring.posSuperimposed := FALSE;
   cmAnodeMainPnP2AxisX.monitoring.haltSuperimposed := FALSE;
   cmAnodeMainPnP2AxisX.monitoring.brakeOpened := FALSE;
   cmAnodeMainPnP2AxisX.monitoring.axisEnabled := TRUE;
   cmAnodeMainPnP2AxisX.monitoring.resetActive := FALSE;
   cmAnodeMainPnP2AxisX.monitoring.inVelocity := FALSE;
   cmAnodeMainPnP2AxisX.monitoring.inLimitation := FALSE;
   cmAnodeMainPnP2AxisX.monitoring.inClamping := FALSE;
   cmAnodeMainPnP2AxisX.monitoring.startSync := FALSE;
   cmAnodeMainPnP2AxisX.monitoring.inSync := FALSE;
   cmAnodeMainPnP2AxisX.monitoring.inSimulation := FALSE;
   cmAnodeMainPnP2AxisX.monitoring.jogSelected := FALSE;
   cmAnodeMainPnP2AxisX.monitoring.moveVelocitySelected := FALSE;
   cmAnodeMainPnP2AxisX.monitoring.stopSelected := FALSE;
   cmAnodeMainPnP2AxisX.monitoring.fastStopSelected := FALSE;
   cmAnodeMainPnP2AxisX.monitoring.torqueLimitingSelected := FALSE;
   cmAnodeMainPnP2AxisX.monitoring.homingSelected := FALSE;
   cmAnodeMainPnP2AxisX.monitoring.posRelativeSelected := FALSE;
   cmAnodeMainPnP2AxisX.monitoring.posAbsoluteSelected := FALSE;
   cmAnodeMainPnP2AxisX.monitoring.posSuperimposedSelected := FALSE;
   cmAnodeMainPnP2AxisX.monitoring.haltSuperimposedSelected := FALSE;
   cmAnodeMainPnP2AxisX.monitoring.commandBusy := FALSE;
   cmAnodeMainPnP2AxisX.monitoring.commandDone := FALSE;
   cmAnodeMainPnP2AxisX.monitoring.commandAborted := FALSE;
   cmAnodeMainPnP2AxisX.monitoring.homingCommandBusy := FALSE;
   cmAnodeMainPnP2AxisX.monitoring.homingCommandDone := FALSE;
   cmAnodeMainPnP2AxisX.monitoring.homingCommandAborted := FALSE;
   cmAnodeMainPnP2AxisX.monitoring.superimposedBusy := FALSE;
   cmAnodeMainPnP2AxisX.monitoring.superimposedDone := FALSE;
   cmAnodeMainPnP2AxisX.monitoring.superimposedAborted := FALSE;
   cmAnodeMainPnP2AxisX.monitoring.selectSetPosition := 1;
   cmAnodeMainPnP2AxisX.monitoring.selectionController := FALSE;
   cmAnodeMainPnP2AxisX.monitoring.interlockGeneral := TRUE;
   cmAnodeMainPnP2AxisX.monitoring.interlockJogForward := TRUE;
   cmAnodeMainPnP2AxisX.monitoring.interlockJogBackward := TRUE;
   cmAnodeMainPnP2AxisX.monitoring.interlockWarningGeneral := FALSE;
   cmAnodeMainPnP2AxisX.monitoring.interlockWarningJogForward := FALSE;
   cmAnodeMainPnP2AxisX.monitoring.interlockWarningJogBackward := FALSE;
   cmAnodeMainPnP2AxisX.monitoring.valid := TRUE;
   cmAnodeMainPnP2AxisX.monitoring.busy := TRUE;
   cmAnodeMainPnP2AxisX.monitoring.error := FALSE;
   cmAnodeMainPnP2AxisX.monitoring.status := 16#7002;
   cmAnodeMainPnP2AxisX.monitoring.subfunctionStatus := 16#0000;
   cmAnodeMainPnP2AxisX.monitoring.actualPosition := 539.98;
   cmAnodeMainPnP2AxisX.monitoring.actualSpeed := 6.62553364956176;
   cmAnodeMainPnP2AxisX.monitoring.speedUnit := 1062;
   cmAnodeMainPnP2AxisX.monitoring.positionUnit := 1013;
   cmAnodeMainPnP2AxisX.monitoring.axisStatus1 := 16#0240_4021;
   cmAnodeMainPnP2AxisX.monitoring.axisStatus2 := 16#0000_0000;
   cmAnodeMainPnP2AxisX.monitoring.axisType := 1;
   cmAnodeMainPnP2AxisX.monitoring.maxVelocity := 2500.0;
   cmAnodeMainPnP2AxisX.monitoring.actualCurrent := 0.0;
   cmAnodeMainPnP2AxisX.monitoring.actualTorque := 0.0;
   cmAnodeMainPnP2AxisX.monitoring.velocityOverrideEnabled := FALSE;
   cmAnodeMainPnP2AxisX.monitoring.sinaParaError := FALSE;
   cmAnodeMainPnP2AxisX.monitoring.sinaParaStatus := 16#0000_0000;
   cmAnodeMainPnP2AxisX.configuration.referenceDesignator := WSTRING#'AnodeMainPnP2AxisX';
   cmAnodeMainPnP2AxisX.configuration.disableAlarms := FALSE;
   cmAnodeMainPnP2AxisX.configuration.masterControlPopUp := TRUE;
   cmAnodeMainPnP2AxisX.configuration.setPositions[0].position := 540.0;
   cmAnodeMainPnP2AxisX.configuration.setPositions[1].position := 0.0;
   cmAnodeMainPnP2AxisX.configuration.setPositions[2].position := -3.5;
   cmAnodeMainPnP2AxisX.configuration.setPositions[3..15].position := 0.0;
   cmAnodeMainPnP2AxisX.configuration.setPositions[0..1].velocity := 500.0;
   cmAnodeMainPnP2AxisX.configuration.setPositions[2].velocity := 100.0;
   cmAnodeMainPnP2AxisX.configuration.setPositions[3..15].velocity := -1.0;
   cmAnodeMainPnP2AxisX.configuration.setPositions[0..1].acceleration := 5000.0;
   cmAnodeMainPnP2AxisX.configuration.setPositions[2].acceleration := 30.0;
   cmAnodeMainPnP2AxisX.configuration.setPositions[3..15].acceleration := -1.0;
   cmAnodeMainPnP2AxisX.configuration.setPositions[0..1].deceleration := 5000.0;
   cmAnodeMainPnP2AxisX.configuration.setPositions[2].deceleration := 30.0;
   cmAnodeMainPnP2AxisX.configuration.setPositions[3..15].deceleration := -1.0;
   cmAnodeMainPnP2AxisX.configuration.setPositions[0..15]."name" := '';
   cmAnodeMainPnP1AxisY.commandConfiguration.generalSettings.stopOnError := TRUE;
   cmAnodeMainPnP1AxisY.commandConfiguration.generalSettings.resetWithRestart := FALSE;
   cmAnodeMainPnP1AxisY.commandConfiguration.generalSettings.abortWaitingSyncCmd := TRUE;
   cmAnodeMainPnP1AxisY.commandConfiguration.power.startMode := 1;
   cmAnodeMainPnP1AxisY.commandConfiguration.power.stopMode := 0;
   cmAnodeMainPnP1AxisY.commandConfiguration.power.syncMotionSimulation := FALSE;
   cmAnodeMainPnP1AxisY.commandConfiguration.power.syncMotionSimulationExtendedMode := -1;
   cmAnodeMainPnP1AxisY.commandConfiguration.jog.velocity := 10.0;
   cmAnodeMainPnP1AxisY.commandConfiguration.jog.acceleration := 100.0;
   cmAnodeMainPnP1AxisY.commandConfiguration.jog.deceleration := 100.0;
   cmAnodeMainPnP1AxisY.commandConfiguration.jog.jerk := -1.0;
   cmAnodeMainPnP1AxisY.commandConfiguration.jog.positionControlled := TRUE;
   cmAnodeMainPnP1AxisY.commandConfiguration.jog.increment := 0.0;
   cmAnodeMainPnP1AxisY.commandConfiguration.jog.mode := 0;
   cmAnodeMainPnP1AxisY.commandConfiguration.moveVelocity.velocity := 10.0;
   cmAnodeMainPnP1AxisY.commandConfiguration.moveVelocity.acceleration := 100.0;
   cmAnodeMainPnP1AxisY.commandConfiguration.moveVelocity.deceleration := 100.0;
   cmAnodeMainPnP1AxisY.commandConfiguration.moveVelocity.jerk := -1.0;
   cmAnodeMainPnP1AxisY.commandConfiguration.moveVelocity.direction := 0;
   cmAnodeMainPnP1AxisY.commandConfiguration.moveVelocity.positionControlled := TRUE;
   cmAnodeMainPnP1AxisY.commandConfiguration.moveVelocity.velocityChangeOnTheFly := FALSE;
   cmAnodeMainPnP1AxisY.commandConfiguration.stop.deceleration := -1.0;
   cmAnodeMainPnP1AxisY.commandConfiguration.stop.jerk := -1.0;
   cmAnodeMainPnP1AxisY.commandConfiguration.stop.abortAcceleration := FALSE;
   cmAnodeMainPnP1AxisY.commandConfiguration.fastStop.deceleration := -1.0;
   cmAnodeMainPnP1AxisY.commandConfiguration.fastStop.jerk := -1.0;
   cmAnodeMainPnP1AxisY.commandConfiguration.fastStop.abortAcceleration := FALSE;
   cmAnodeMainPnP1AxisY.commandConfiguration.fastStop.replaceStopPossible := FALSE;
   cmAnodeMainPnP1AxisY.commandConfiguration.torqueLimiting.limit := -1.0;
   cmAnodeMainPnP1AxisY.commandConfiguration.torqueLimiting.mode := 0;
   cmAnodeMainPnP1AxisY.commandConfiguration.homing.position := 0.0;
   cmAnodeMainPnP1AxisY.commandConfiguration.homing.mode := 0;
   cmAnodeMainPnP1AxisY.commandConfiguration.homing.sensor := 0;
   cmAnodeMainPnP1AxisY.commandConfiguration.homing.extendedMode := -1;
   cmAnodeMainPnP1AxisY.commandConfiguration.homing.extendedModeTorqueLimit := 0.0;
   cmAnodeMainPnP1AxisY.commandConfiguration.homing.extendedModeTargetPosition := 0.0;
   cmAnodeMainPnP1AxisY.commandConfiguration.posRelative.distance := 0.0;
   cmAnodeMainPnP1AxisY.commandConfiguration.posRelative.velocity := 10.0;
   cmAnodeMainPnP1AxisY.commandConfiguration.posRelative.acceleration := 100.0;
   cmAnodeMainPnP1AxisY.commandConfiguration.posRelative.deceleration := 100.0;
   cmAnodeMainPnP1AxisY.commandConfiguration.posRelative.jerk := -1.0;
   cmAnodeMainPnP1AxisY.commandConfiguration.posRelative.direction := 0;
   cmAnodeMainPnP1AxisY.commandConfiguration.posAbsolute.position := 0.0;
   cmAnodeMainPnP1AxisY.commandConfiguration.posAbsolute.velocity := -1.0;
   cmAnodeMainPnP1AxisY.commandConfiguration.posAbsolute.acceleration := -1.0;
   cmAnodeMainPnP1AxisY.commandConfiguration.posAbsolute.deceleration := -1.0;
   cmAnodeMainPnP1AxisY.commandConfiguration.posAbsolute.jerk := -1.0;
   cmAnodeMainPnP1AxisY.commandConfiguration.posAbsolute.direction := 1;
   cmAnodeMainPnP1AxisY.commandConfiguration.posAbsolute.positionChangeOnTheFly := FALSE;
   cmAnodeMainPnP1AxisY.commandConfiguration.posAbsolute.velocityChangeOnTheFly := FALSE;
   cmAnodeMainPnP1AxisY.commandConfiguration.posSuperimposed.distance := 0.0;
   cmAnodeMainPnP1AxisY.commandConfiguration.posSuperimposed.velocityDiff := -1.0;
   cmAnodeMainPnP1AxisY.commandConfiguration.posSuperimposed.acceleration := -1.0;
   cmAnodeMainPnP1AxisY.commandConfiguration.posSuperimposed.deceleration := -1.0;
   cmAnodeMainPnP1AxisY.commandConfiguration.posSuperimposed.jerk := -1.0;
   cmAnodeMainPnP1AxisY.commandConfiguration.posSuperimposed.direction := 0;
   cmAnodeMainPnP1AxisY.commandConfiguration.haltSuperimposed.deceleration := -1.0;
   cmAnodeMainPnP1AxisY.commandConfiguration.haltSuperimposed.jerk := -1.0;
   cmAnodeMainPnP1AxisY.commandConfiguration.haltSuperimposed.abortAcceleration := FALSE;
   cmAnodeMainPnP1AxisY.commandConfiguration.gearInRelative.ratioNumerator := 1;
   cmAnodeMainPnP1AxisY.commandConfiguration.gearInRelative.ratioDenominator := 1;
   cmAnodeMainPnP1AxisY.commandConfiguration.gearInRelative.acceleration := -1.0;
   cmAnodeMainPnP1AxisY.commandConfiguration.gearInRelative.deceleration := -1.0;
   cmAnodeMainPnP1AxisY.commandConfiguration.gearInRelative.jerk := -1.0;
   cmAnodeMainPnP1AxisY.commandConfiguration.gearInRelative.ratioChangeOnTheFly := FALSE;
   cmAnodeMainPnP1AxisY.commandConfiguration.gearInAbsolute.ratioNumerator := 1;
   cmAnodeMainPnP1AxisY.commandConfiguration.gearInAbsolute.ratioDenominator := 1;
   cmAnodeMainPnP1AxisY.commandConfiguration.gearInAbsolute.masterSyncPosition := 0.0;
   cmAnodeMainPnP1AxisY.commandConfiguration.gearInAbsolute.slaveSyncPosition := 0.0;
   cmAnodeMainPnP1AxisY.commandConfiguration.gearInAbsolute.syncProfileReference := 1;
   cmAnodeMainPnP1AxisY.commandConfiguration.gearInAbsolute.masterStartDistance := 0.0;
   cmAnodeMainPnP1AxisY.commandConfiguration.gearInAbsolute.velocity := -1.0;
   cmAnodeMainPnP1AxisY.commandConfiguration.gearInAbsolute.acceleration := -1.0;
   cmAnodeMainPnP1AxisY.commandConfiguration.gearInAbsolute.deceleration := -1.0;
   cmAnodeMainPnP1AxisY.commandConfiguration.gearInAbsolute.jerk := -1.0;
   cmAnodeMainPnP1AxisY.commandConfiguration.gearInAbsolute.syncDirection := 1;
   cmAnodeMainPnP1AxisY.commandConfiguration.gearInAbsolute.ratioChangeOnTheFly := FALSE;
   cmAnodeMainPnP1AxisY.commandConfiguration.gearInVelocity.continuousUpdate := FALSE;
   cmAnodeMainPnP1AxisY.commandConfiguration.gearInVelocity.ratioNumerator := 1;
   cmAnodeMainPnP1AxisY.commandConfiguration.gearInVelocity.ratioDenominator := 1;
   cmAnodeMainPnP1AxisY.commandConfiguration.gearInVelocity.acceleration := -1.0;
   cmAnodeMainPnP1AxisY.commandConfiguration.gearInVelocity.deceleration := -1.0;
   cmAnodeMainPnP1AxisY.commandConfiguration.gearInVelocity.jerk := -1.0;
   cmAnodeMainPnP1AxisY.commandConfiguration.gearInVelocity.positionControlled := FALSE;
   cmAnodeMainPnP1AxisY.commandConfiguration.camIn.masterOffset := 0.0;
   cmAnodeMainPnP1AxisY.commandConfiguration.camIn.slaveOffset := 0.0;
   cmAnodeMainPnP1AxisY.commandConfiguration.camIn.masterScaling := 1.0;
   cmAnodeMainPnP1AxisY.commandConfiguration.camIn.slaveScaling := 1.0;
   cmAnodeMainPnP1AxisY.commandConfiguration.camIn.masterSyncPosition := 0.0;
   cmAnodeMainPnP1AxisY.commandConfiguration.camIn.syncProfileReference := 1;
   cmAnodeMainPnP1AxisY.commandConfiguration.camIn.masterStartDistance := 0.0;
   cmAnodeMainPnP1AxisY.commandConfiguration.camIn.velocity := -1.0;
   cmAnodeMainPnP1AxisY.commandConfiguration.camIn.acceleration := -1.0;
   cmAnodeMainPnP1AxisY.commandConfiguration.camIn.deceleration := -1.0;
   cmAnodeMainPnP1AxisY.commandConfiguration.camIn.jerk := -1.0;
   cmAnodeMainPnP1AxisY.commandConfiguration.camIn.applicationMode := 0;
   cmAnodeMainPnP1AxisY.commandConfiguration.camIn.syncDirection := 1;
   cmAnodeMainPnP1AxisY.commandConfiguration.gearOutCamOut.slavePosition := 0.0;
   cmAnodeMainPnP1AxisY.commandConfiguration.gearOutCamOut.syncProfileReference := 1;
   cmAnodeMainPnP1AxisY.commandConfiguration.gearOutCamOut.masterStopDistance := 0.0;
   cmAnodeMainPnP1AxisY.commandConfiguration.gearOutCamOut.deceleration := -1.0;
   cmAnodeMainPnP1AxisY.commandConfiguration.gearOutCamOut.jerk := -1.0;
   cmAnodeMainPnP1AxisY.commandConfiguration.gearOutCamOut.syncOutDirection := 3;
   cmAnodeMainPnP1AxisY.commandConfiguration.gearOutCamOut.gearOutCamOutMode := -1;
   cmAnodeMainPnP1AxisY.commandConfiguration.phasing.phaseShift := 0.0;
   cmAnodeMainPnP1AxisY.commandConfiguration.phasing.velocity := -1.0;
   cmAnodeMainPnP1AxisY.commandConfiguration.phasing.acceleration := -1.0;
   cmAnodeMainPnP1AxisY.commandConfiguration.phasing.deceleration := -1.0;
   cmAnodeMainPnP1AxisY.commandConfiguration.phasing.jerk := -1.0;
   cmAnodeMainPnP1AxisY.commandConfiguration.phasing.profileReference := 0;
   cmAnodeMainPnP1AxisY.commandConfiguration.phasing.phasingDistance := 0.0;
   cmAnodeMainPnP1AxisY.commandConfiguration.phasing.startPosition := 0.0;
   cmAnodeMainPnP1AxisY.commandConfiguration.phasing.direction := 3;
   cmAnodeMainPnP1AxisY.commandConfiguration.phasing.phaseAbsolute := TRUE;
   cmAnodeMainPnP1AxisY.commandConfiguration.phasing.phaseShiftChangeOnTheFly := FALSE;
   cmAnodeMainPnP1AxisY.commandConfiguration.offset.offset := 0.0;
   cmAnodeMainPnP1AxisY.commandConfiguration.offset.profileReference := 1;
   cmAnodeMainPnP1AxisY.commandConfiguration.offset.offsetDistance := 0.0;
   cmAnodeMainPnP1AxisY.commandConfiguration.offset.startPosition := 0.0;
   cmAnodeMainPnP1AxisY.commandConfiguration.offset.direction := 3;
   cmAnodeMainPnP1AxisY.commandConfiguration.offset.offsetAbsolute := TRUE;
   cmAnodeMainPnP1AxisY.commandConfiguration.offset.offsetChangeOnTheFly := FALSE;
   cmAnodeMainPnP1AxisY.commands.enableMasterControl := TRUE;
   cmAnodeMainPnP1AxisY.commands.enableAxis := FALSE;
   cmAnodeMainPnP1AxisY.commands.resetAxis := FALSE;
   cmAnodeMainPnP1AxisY.commands.openBrake := FALSE;
   cmAnodeMainPnP1AxisY.commands.jogForward := FALSE;
   cmAnodeMainPnP1AxisY.commands.jogBackward := FALSE;
   cmAnodeMainPnP1AxisY.commands.moveVelocity := FALSE;
   cmAnodeMainPnP1AxisY.commands.stop := FALSE;
   cmAnodeMainPnP1AxisY.commands.fastStop := FALSE;
   cmAnodeMainPnP1AxisY.commands.torqueLimiting := FALSE;
   cmAnodeMainPnP1AxisY.commands.homing := FALSE;
   cmAnodeMainPnP1AxisY.commands.posRelative := FALSE;
   cmAnodeMainPnP1AxisY.commands.posAbsolute := FALSE;
   cmAnodeMainPnP1AxisY.commands.posSuperimposed := FALSE;
   cmAnodeMainPnP1AxisY.commands.haltSuperimposed := FALSE;
   cmAnodeMainPnP1AxisY.commands.selectSetPosition := -1;
   cmAnodeMainPnP1AxisY.commands.uploadParameters := FALSE;
   cmAnodeMainPnP1AxisY.commands.refreshConfiguration := FALSE;
   cmAnodeMainPnP1AxisY.commands.editConfiguration := FALSE;
   cmAnodeMainPnP1AxisY.commands.saveConfiguration := FALSE;
   cmAnodeMainPnP1AxisY.commands.uploadCurrentTorque := FALSE;
   cmAnodeMainPnP1AxisY.commands.reset := FALSE;
   cmAnodeMainPnP1AxisY.monitoring.enable := TRUE;
   cmAnodeMainPnP1AxisY.monitoring.referenceDesignator := WSTRING#'AnodeMainPnP1AxisY';
   cmAnodeMainPnP1AxisY.monitoring.enabled := TRUE;
   cmAnodeMainPnP1AxisY.monitoring.enableManualCmds := FALSE;
   cmAnodeMainPnP1AxisY.monitoring.reset := FALSE;
   cmAnodeMainPnP1AxisY.monitoring.resetAxis := FALSE;
   cmAnodeMainPnP1AxisY.monitoring.enableAxis := TRUE;
   cmAnodeMainPnP1AxisY.monitoring.openBrake := FALSE;
   cmAnodeMainPnP1AxisY.monitoring.jogBackward := FALSE;
   cmAnodeMainPnP1AxisY.monitoring.jogForward := FALSE;
   cmAnodeMainPnP1AxisY.monitoring.moveVelocity := FALSE;
   cmAnodeMainPnP1AxisY.monitoring.stop := FALSE;
   cmAnodeMainPnP1AxisY.monitoring.fastStop := FALSE;
   cmAnodeMainPnP1AxisY.monitoring.torqueLimiting := FALSE;
   cmAnodeMainPnP1AxisY.monitoring.homing := FALSE;
   cmAnodeMainPnP1AxisY.monitoring.posRelative := FALSE;
   cmAnodeMainPnP1AxisY.monitoring.posAbsolute := FALSE;
   cmAnodeMainPnP1AxisY.monitoring.posSuperimposed := FALSE;
   cmAnodeMainPnP1AxisY.monitoring.haltSuperimposed := FALSE;
   cmAnodeMainPnP1AxisY.monitoring.brakeOpened := FALSE;
   cmAnodeMainPnP1AxisY.monitoring.axisEnabled := TRUE;
   cmAnodeMainPnP1AxisY.monitoring.resetActive := FALSE;
   cmAnodeMainPnP1AxisY.monitoring.inVelocity := FALSE;
   cmAnodeMainPnP1AxisY.monitoring.inLimitation := FALSE;
   cmAnodeMainPnP1AxisY.monitoring.inClamping := FALSE;
   cmAnodeMainPnP1AxisY.monitoring.startSync := FALSE;
   cmAnodeMainPnP1AxisY.monitoring.inSync := FALSE;
   cmAnodeMainPnP1AxisY.monitoring.inSimulation := FALSE;
   cmAnodeMainPnP1AxisY.monitoring.jogSelected := FALSE;
   cmAnodeMainPnP1AxisY.monitoring.moveVelocitySelected := FALSE;
   cmAnodeMainPnP1AxisY.monitoring.stopSelected := FALSE;
   cmAnodeMainPnP1AxisY.monitoring.fastStopSelected := FALSE;
   cmAnodeMainPnP1AxisY.monitoring.torqueLimitingSelected := FALSE;
   cmAnodeMainPnP1AxisY.monitoring.homingSelected := FALSE;
   cmAnodeMainPnP1AxisY.monitoring.posRelativeSelected := FALSE;
   cmAnodeMainPnP1AxisY.monitoring.posAbsoluteSelected := FALSE;
   cmAnodeMainPnP1AxisY.monitoring.posSuperimposedSelected := FALSE;
   cmAnodeMainPnP1AxisY.monitoring.haltSuperimposedSelected := FALSE;
   cmAnodeMainPnP1AxisY.monitoring.commandBusy := FALSE;
   cmAnodeMainPnP1AxisY.monitoring.commandDone := FALSE;
   cmAnodeMainPnP1AxisY.monitoring.commandAborted := FALSE;
   cmAnodeMainPnP1AxisY.monitoring.homingCommandBusy := FALSE;
   cmAnodeMainPnP1AxisY.monitoring.homingCommandDone := FALSE;
   cmAnodeMainPnP1AxisY.monitoring.homingCommandAborted := FALSE;
   cmAnodeMainPnP1AxisY.monitoring.superimposedBusy := FALSE;
   cmAnodeMainPnP1AxisY.monitoring.superimposedDone := FALSE;
   cmAnodeMainPnP1AxisY.monitoring.superimposedAborted := FALSE;
   cmAnodeMainPnP1AxisY.monitoring.selectSetPosition := -1;
   cmAnodeMainPnP1AxisY.monitoring.selectionController := FALSE;
   cmAnodeMainPnP1AxisY.monitoring.interlockGeneral := TRUE;
   cmAnodeMainPnP1AxisY.monitoring.interlockJogForward := TRUE;
   cmAnodeMainPnP1AxisY.monitoring.interlockJogBackward := TRUE;
   cmAnodeMainPnP1AxisY.monitoring.interlockWarningGeneral := FALSE;
   cmAnodeMainPnP1AxisY.monitoring.interlockWarningJogForward := FALSE;
   cmAnodeMainPnP1AxisY.monitoring.interlockWarningJogBackward := FALSE;
   cmAnodeMainPnP1AxisY.monitoring.valid := TRUE;
   cmAnodeMainPnP1AxisY.monitoring.busy := TRUE;
   cmAnodeMainPnP1AxisY.monitoring.error := FALSE;
   cmAnodeMainPnP1AxisY.monitoring.status := 16#7002;
   cmAnodeMainPnP1AxisY.monitoring.subfunctionStatus := 16#0000;
   cmAnodeMainPnP1AxisY.monitoring.actualPosition := 0.0;
   cmAnodeMainPnP1AxisY.monitoring.actualSpeed := 0.0;
   cmAnodeMainPnP1AxisY.monitoring.speedUnit := 1062;
   cmAnodeMainPnP1AxisY.monitoring.positionUnit := 1013;
   cmAnodeMainPnP1AxisY.monitoring.axisStatus1 := 16#0200_10E1;
   cmAnodeMainPnP1AxisY.monitoring.axisStatus2 := 16#0000_0000;
   cmAnodeMainPnP1AxisY.monitoring.axisType := 1;
   cmAnodeMainPnP1AxisY.monitoring.maxVelocity := 2500.0;
   cmAnodeMainPnP1AxisY.monitoring.actualCurrent := 0.0;
   cmAnodeMainPnP1AxisY.monitoring.actualTorque := 0.0;
   cmAnodeMainPnP1AxisY.monitoring.velocityOverrideEnabled := FALSE;
   cmAnodeMainPnP1AxisY.monitoring.sinaParaError := FALSE;
   cmAnodeMainPnP1AxisY.monitoring.sinaParaStatus := 16#0000_0000;
   cmAnodeMainPnP1AxisY.configuration.referenceDesignator := WSTRING#'AnodeMainPnP1AxisY';
   cmAnodeMainPnP1AxisY.configuration.disableAlarms := FALSE;
   cmAnodeMainPnP1AxisY.configuration.masterControlPopUp := TRUE;
   cmAnodeMainPnP1AxisY.configuration.setPositions[0..15].position := 0.0;
   cmAnodeMainPnP1AxisY.configuration.setPositions[0].velocity := 50.0;
   cmAnodeMainPnP1AxisY.configuration.setPositions[1].velocity := 30.0;
   cmAnodeMainPnP1AxisY.configuration.setPositions[2..15].velocity := -1.0;
   cmAnodeMainPnP1AxisY.configuration.setPositions[0].acceleration := 500.0;
   cmAnodeMainPnP1AxisY.configuration.setPositions[1].acceleration := 30.0;
   cmAnodeMainPnP1AxisY.configuration.setPositions[2..15].acceleration := -1.0;
   cmAnodeMainPnP1AxisY.configuration.setPositions[0].deceleration := 500.0;
   cmAnodeMainPnP1AxisY.configuration.setPositions[1].deceleration := 30.0;
   cmAnodeMainPnP1AxisY.configuration.setPositions[2..15].deceleration := -1.0;
   cmAnodeMainPnP1AxisY.configuration.setPositions[0..15]."name" := '';
   cmAnodeMainPnP1AxisZ.commandConfiguration.generalSettings.stopOnError := TRUE;
   cmAnodeMainPnP1AxisZ.commandConfiguration.generalSettings.resetWithRestart := FALSE;
   cmAnodeMainPnP1AxisZ.commandConfiguration.generalSettings.abortWaitingSyncCmd := TRUE;
   cmAnodeMainPnP1AxisZ.commandConfiguration.power.startMode := 1;
   cmAnodeMainPnP1AxisZ.commandConfiguration.power.stopMode := 0;
   cmAnodeMainPnP1AxisZ.commandConfiguration.power.syncMotionSimulation := FALSE;
   cmAnodeMainPnP1AxisZ.commandConfiguration.power.syncMotionSimulationExtendedMode := -1;
   cmAnodeMainPnP1AxisZ.commandConfiguration.jog.velocity := 10.0;
   cmAnodeMainPnP1AxisZ.commandConfiguration.jog.acceleration := 100.0;
   cmAnodeMainPnP1AxisZ.commandConfiguration.jog.deceleration := 100.0;
   cmAnodeMainPnP1AxisZ.commandConfiguration.jog.jerk := -1.0;
   cmAnodeMainPnP1AxisZ.commandConfiguration.jog.positionControlled := TRUE;
   cmAnodeMainPnP1AxisZ.commandConfiguration.jog.increment := 0.0;
   cmAnodeMainPnP1AxisZ.commandConfiguration.jog.mode := 0;
   cmAnodeMainPnP1AxisZ.commandConfiguration.moveVelocity.velocity := 10.0;
   cmAnodeMainPnP1AxisZ.commandConfiguration.moveVelocity.acceleration := 100.0;
   cmAnodeMainPnP1AxisZ.commandConfiguration.moveVelocity.deceleration := 100.0;
   cmAnodeMainPnP1AxisZ.commandConfiguration.moveVelocity.jerk := -1.0;
   cmAnodeMainPnP1AxisZ.commandConfiguration.moveVelocity.direction := 0;
   cmAnodeMainPnP1AxisZ.commandConfiguration.moveVelocity.positionControlled := TRUE;
   cmAnodeMainPnP1AxisZ.commandConfiguration.moveVelocity.velocityChangeOnTheFly := FALSE;
   cmAnodeMainPnP1AxisZ.commandConfiguration.stop.deceleration := -1.0;
   cmAnodeMainPnP1AxisZ.commandConfiguration.stop.jerk := -1.0;
   cmAnodeMainPnP1AxisZ.commandConfiguration.stop.abortAcceleration := FALSE;
   cmAnodeMainPnP1AxisZ.commandConfiguration.fastStop.deceleration := -1.0;
   cmAnodeMainPnP1AxisZ.commandConfiguration.fastStop.jerk := -1.0;
   cmAnodeMainPnP1AxisZ.commandConfiguration.fastStop.abortAcceleration := FALSE;
   cmAnodeMainPnP1AxisZ.commandConfiguration.fastStop.replaceStopPossible := FALSE;
   cmAnodeMainPnP1AxisZ.commandConfiguration.torqueLimiting.limit := -1.0;
   cmAnodeMainPnP1AxisZ.commandConfiguration.torqueLimiting.mode := 0;
   cmAnodeMainPnP1AxisZ.commandConfiguration.homing.position := 0.0;
   cmAnodeMainPnP1AxisZ.commandConfiguration.homing.mode := 0;
   cmAnodeMainPnP1AxisZ.commandConfiguration.homing.sensor := 0;
   cmAnodeMainPnP1AxisZ.commandConfiguration.homing.extendedMode := -1;
   cmAnodeMainPnP1AxisZ.commandConfiguration.homing.extendedModeTorqueLimit := 0.0;
   cmAnodeMainPnP1AxisZ.commandConfiguration.homing.extendedModeTargetPosition := 0.0;
   cmAnodeMainPnP1AxisZ.commandConfiguration.posRelative.distance := 0.0;
   cmAnodeMainPnP1AxisZ.commandConfiguration.posRelative.velocity := 10.0;
   cmAnodeMainPnP1AxisZ.commandConfiguration.posRelative.acceleration := 100.0;
   cmAnodeMainPnP1AxisZ.commandConfiguration.posRelative.deceleration := 100.0;
   cmAnodeMainPnP1AxisZ.commandConfiguration.posRelative.jerk := -1.0;
   cmAnodeMainPnP1AxisZ.commandConfiguration.posRelative.direction := 0;
   cmAnodeMainPnP1AxisZ.commandConfiguration.posAbsolute.position := 0.0;
   cmAnodeMainPnP1AxisZ.commandConfiguration.posAbsolute.velocity := -1.0;
   cmAnodeMainPnP1AxisZ.commandConfiguration.posAbsolute.acceleration := -1.0;
   cmAnodeMainPnP1AxisZ.commandConfiguration.posAbsolute.deceleration := -1.0;
   cmAnodeMainPnP1AxisZ.commandConfiguration.posAbsolute.jerk := -1.0;
   cmAnodeMainPnP1AxisZ.commandConfiguration.posAbsolute.direction := 1;
   cmAnodeMainPnP1AxisZ.commandConfiguration.posAbsolute.positionChangeOnTheFly := FALSE;
   cmAnodeMainPnP1AxisZ.commandConfiguration.posAbsolute.velocityChangeOnTheFly := FALSE;
   cmAnodeMainPnP1AxisZ.commandConfiguration.posSuperimposed.distance := 0.0;
   cmAnodeMainPnP1AxisZ.commandConfiguration.posSuperimposed.velocityDiff := -1.0;
   cmAnodeMainPnP1AxisZ.commandConfiguration.posSuperimposed.acceleration := -1.0;
   cmAnodeMainPnP1AxisZ.commandConfiguration.posSuperimposed.deceleration := -1.0;
   cmAnodeMainPnP1AxisZ.commandConfiguration.posSuperimposed.jerk := -1.0;
   cmAnodeMainPnP1AxisZ.commandConfiguration.posSuperimposed.direction := 0;
   cmAnodeMainPnP1AxisZ.commandConfiguration.haltSuperimposed.deceleration := -1.0;
   cmAnodeMainPnP1AxisZ.commandConfiguration.haltSuperimposed.jerk := -1.0;
   cmAnodeMainPnP1AxisZ.commandConfiguration.haltSuperimposed.abortAcceleration := FALSE;
   cmAnodeMainPnP1AxisZ.commandConfiguration.gearInRelative.ratioNumerator := 1;
   cmAnodeMainPnP1AxisZ.commandConfiguration.gearInRelative.ratioDenominator := 1;
   cmAnodeMainPnP1AxisZ.commandConfiguration.gearInRelative.acceleration := -1.0;
   cmAnodeMainPnP1AxisZ.commandConfiguration.gearInRelative.deceleration := -1.0;
   cmAnodeMainPnP1AxisZ.commandConfiguration.gearInRelative.jerk := -1.0;
   cmAnodeMainPnP1AxisZ.commandConfiguration.gearInRelative.ratioChangeOnTheFly := FALSE;
   cmAnodeMainPnP1AxisZ.commandConfiguration.gearInAbsolute.ratioNumerator := 1;
   cmAnodeMainPnP1AxisZ.commandConfiguration.gearInAbsolute.ratioDenominator := 1;
   cmAnodeMainPnP1AxisZ.commandConfiguration.gearInAbsolute.masterSyncPosition := 0.0;
   cmAnodeMainPnP1AxisZ.commandConfiguration.gearInAbsolute.slaveSyncPosition := 0.0;
   cmAnodeMainPnP1AxisZ.commandConfiguration.gearInAbsolute.syncProfileReference := 1;
   cmAnodeMainPnP1AxisZ.commandConfiguration.gearInAbsolute.masterStartDistance := 0.0;
   cmAnodeMainPnP1AxisZ.commandConfiguration.gearInAbsolute.velocity := -1.0;
   cmAnodeMainPnP1AxisZ.commandConfiguration.gearInAbsolute.acceleration := -1.0;
   cmAnodeMainPnP1AxisZ.commandConfiguration.gearInAbsolute.deceleration := -1.0;
   cmAnodeMainPnP1AxisZ.commandConfiguration.gearInAbsolute.jerk := -1.0;
   cmAnodeMainPnP1AxisZ.commandConfiguration.gearInAbsolute.syncDirection := 1;
   cmAnodeMainPnP1AxisZ.commandConfiguration.gearInAbsolute.ratioChangeOnTheFly := FALSE;
   cmAnodeMainPnP1AxisZ.commandConfiguration.gearInVelocity.continuousUpdate := FALSE;
   cmAnodeMainPnP1AxisZ.commandConfiguration.gearInVelocity.ratioNumerator := 1;
   cmAnodeMainPnP1AxisZ.commandConfiguration.gearInVelocity.ratioDenominator := 1;
   cmAnodeMainPnP1AxisZ.commandConfiguration.gearInVelocity.acceleration := -1.0;
   cmAnodeMainPnP1AxisZ.commandConfiguration.gearInVelocity.deceleration := -1.0;
   cmAnodeMainPnP1AxisZ.commandConfiguration.gearInVelocity.jerk := -1.0;
